// ---- DUTs/EPS Robot/CmdRobot1.TcDUT
{attribute 'qualified_only'}
{attribute 'strict'}
TYPE CmdRobot1 :
(
	noCmd := 0 ,
	Cmd_GoHome:=1 ,
	Cmd_TakePart:=2 ,
	Cmd_PutPart:=4
	//1=回原点程序  2=取料程序  3=放料程序
	
)WORD;
END_TYPE

// ---- DUTs/EPS Robot/DUT_SysFromRobot1.TcDUT
TYPE DUT_SysFromRobot1 :
STRUCT
//Robot-PLC
xHomePosReached	    		:BOOL;//回原点完成
xPickPartPosReached 	  :BOOL;//到达取料位
xPutPartPosReached			:BOOL;//到达放料位
xPickPos1Reached				:BOOL;//到达主流线取料位置1
xPickPos2Reached				:BOOL;//到达主流线取料位置2
xPickPos3Reached				:BOOL;//到达buffer位置取料
xPickTransferPosReached	:BOOL;//到达中转位置
xPutPos1Reached         :BOOL;//到达皮带线位置1
xPutPos2Reached         :BOOL;//到达皮带线位置2
xPutPos3Reached         :BOOL;//到达NG流道位置
xPutPos4Reached					:BOOL;//到达缓存取料位置

xStepRunning						:BOOL;//子程序已运行
xStepRunDone        		:BOOL;//流程已运行
xInitOK            			:BOOL;//初始化完成
xOutofseg1   						:BOOL;//干涉区1外
xOutofseg2          	  :BOOL;//干涉区2外
xOutofseg3          	  :BOOL;//干涉区3外
END_STRUCT
END_TYPE

// ---- DUTs/EPS Robot/DUT_SysToRobot1.TcDUT
TYPE DUT_SysToRobot1 :
STRUCT
//PLC-Robot	
xStepRunPermit      	:BOOL;//流程允许运行
xClampPartDone				:BOOL;//夹取孔板完成	
xReleasePartDone   		:BOOL;//释放孔板完成
xPickPos1Premit				:BOOL;//去主线位置1取料允许
xPickPos2Premit				:BOOL;//去主线位置2取料允许
xPickPos3Premit				:BOOL;//去buffer位置取料允许
xPickTransferPosPremit:BOOL;//去中转位置允许
xPutPos1Premit				:BOOL;//去皮带线位置1放料允许
xPutPos2Premit				:BOOL;//去皮带线位置2放料允许
xPutPos3Premit				:BOOL;//去NG流道位置放料允许
xPutPos4Premit				:BOOL;//去buffer位置放料允许
iMoveMode           	:WORD;//1=回原点   2=取料程序  4=放料程序
iRatio              	:WORD;//机器人速率
END_STRUCT
END_TYPE

// ---- DUTs/EPS Robot/stPutPartPosChoose.TcDUT
{attribute 'qualified_only'}
{attribute 'strict'}
TYPE stPutPartPosChoose :
(
	enum_member := 0,
	CardPositon_1 := 1,
	CardPostion_2 := 2,
	NGPositon	  :=3,
	BufferPostion :=4
)WORD;
END_TYPE

// ---- DUTs/EPS Robot/stTakePartPosChoose.TcDUT
{attribute 'qualified_only'}
{attribute 'strict'}
TYPE stTakePartPosChoose :
(
	enum_member := 0,
	CardPositon_1 := 1,
	CardPostion_2 := 2,
	BufferPostion :=3
)WORD;
END_TYPE

// ---- DUTs/IO/EL1889.TcDUT
TYPE EL1889 :
STRUCT
	INPUT          :word;
END_STRUCT
END_TYPE

// ---- DUTs/IO/EL2889.TcDUT
TYPE EL2889 :
STRUCT
	OUTPUT          :WORD;
END_STRUCT
END_TYPE

// ---- DUTs/Others/DUT_Calibration.TcDUT
TYPE DUT_Calibration :
STRUCT
	strCalibHmi:STRING;	//校准信息
	xWindowsTrigger :BOOL;//窗口调用
	xStartButtonHmi:BOOL;//校准开始按钮
	xNextButtonHmi:BOOL;//下一组
	xCompletedButtonHmi:BOOL;//校准完成按钮
	xNeedCalibration  :BOOL;//需要校准标志位
	iXCounter:INT;//泵头
	iYCounter:INT;//控制器
	rRudongPumpVolume:REAL;//蠕动泵设定量
	rMckVolume			:REAL;//称测量的量
	rDensity				:REAL;//溶液密度
	iType						:INT:=1;//溶液类型
	iInjectCounter	:INT:=1;//注液次数
	xError  			  :BOOL;//报警
	xReset					:BOOL;//复位报警
END_STRUCT
END_TYPE

// ---- DUTs/Others/DUT_Sta.TcDUT
TYPE DUT_Sta :
STRUCT
		Staion:ARRAY[1..gc_uiStationNum] OF  DUT_StaHistory;
END_STRUCT
END_TYPE

// ---- DUTs/Others/DUT_StaHistory.TcDUT
TYPE DUT_StaHistory :
STRUCT
		History:ARRAY [1..500] OF STRING[100];
END_STRUCT
END_TYPE

// ---- DUTs/Others/stEasyPumpsParamter.TcDUT
TYPE stEasyPumpsParamter :
STRUCT
 		xRdyCmd:BOOL;
		xStart:BOOL;
		xReset:BOOL;
		xBusy:BOOL;
		xError:BOOL;
		xDone:BOOL; 
		
		// 手动校准步骤
		iMCalibStep,iOldMCalibStep: INT;

 		iPumpContorller:INT;
		iPumpModule:INT;
		rSetVolume:REAL;
		rRunTime :REAL;
		iCycleNum:INT;
		iBackAngle:INT;
		rAverageRealVolume:REAL;
		arrRealVolume:ARRAY[1..3] OF REAL;
		arrTestRealVolume:ARRAY[1..50] OF REAL;
		arrRecordVolume:ARRAY[1..50] OF REAL;
		iInjectCounter:INT;
		iCalibCounter:INT;
		iRecordCounter:INT;
		//操作
		
		xModulePushStart:BOOL;//单通道注液开始
		xCalibTestStart:BOOL;//校准测试开始
		xRecordDataStart:BOOL;//记录数据开始
		xModulePushOK:BOOL;//注液OK
		xCalibTestOK:BOOL;//校准测试OK
		xRecordDataOK:BOOL;//记录数据OK
		tStableDelay: TON;
		xInitCalibration:BOOL;//初始化校准系数
		xGotoPosition:BOOL;//去校准位置
		xNeedInjectAgain:BOOL;//需要重新注液
		
		//上下偏差
		rESVolume: REAL;//上偏差
		rEIVolume: REAL;//下偏差
		
END_STRUCT
END_TYPE

// ---- DUTs/Others/stWorkStatus.TcDUT
{attribute 'qualified_only'}
{attribute 'strict'}
TYPE stWorkStatus :
(
	None := 0,
	Started:=1,
	Completed:=2
)BYTE;
END_TYPE

// ---- DUTs/Others/tDateAndTime.TcDUT
TYPE tDateAndTime :
STRUCT

     wYear				: WORD;
     wMonth				: WORD;
     wDayOfWeek	    	: WORD;
     wDay				: WORD;
     wHour				: WORD;
     wMinute			: WORD;
     wSecond			: WORD;
     wMilliseconds 	: WORD;

END_STRUCT
END_TYPE

// ---- DUTs/PartData/DUT_BeltLineFixture.TcDUT
TYPE DUT_BeltLineFixture :
STRUCT
 	xMaterialOnOff : BOOL ;
  stProduct : DUT_PartStatus_1 ;
END_STRUCT
END_TYPE

// ---- DUTs/PartData/DUT_LidChecking.TcDUT
TYPE DUT_LidChecking :
STRUCT
	arCameraResult:ARRAY[1..4,1..12] OF INT;
END_STRUCT
END_TYPE

// ---- DUTs/PartData/DUT_MainlineFixture.TcDUT
TYPE DUT_MainlineFixture :
STRUCT
		xMaterialOnOff : BOOL ;
    stProduct : DUT_PartStatus ;
		stProductFlag :DUT_PartFlag;
		stProcessData:DUT_LidChecking;
		arCycletimeStation: ARRAY[1..20] OF REAL;
END_STRUCT
END_TYPE

// ---- DUTs/PartData/DUT_PartFlag.TcDUT
TYPE DUT_PartFlag :
STRUCT
	xLoading_Bypass :BOOL ;
	xLabeling_Bypass: BOOL ;
	xLidExtracting_Bypass : BOOL ;
	xCoverTightening_Bypass : BOOL ;
	xMarking_Bypass: BOOL ;
	xLabelCheck_Bypass: BOOL ;
	xCoverChcek_Bypass:BOOL;
	
	xNeedChangePallet:BOOL;
	xNeedLabelRepeat :BOOL;
END_STRUCT
END_TYPE

// ---- DUTs/PartData/DUT_PartStatus.TcDUT
TYPE DUT_PartStatus :
STRUCT
	xALL_OK : 	BOOL ; //总的OK
	xPart_Normal :BOOL;//产品正常
	xPart_NG	:BOOL;	//其中有NG
	xLoading_OK :BOOL ;
	xLoading_NOK :BOOL;
	xlidInjecting_OK: BOOL ;
	xlidInjecting_NOK :BOOL;
	xLidChecking_OK : BOOL ;
	xLidChecking_NOK :BOOL;
	xAluCovering_OK : BOOL ;
	xAluCovering_NOK :BOOL;
	xAdjusting_OK: BOOL ;
	xAdjusting_NOK :BOOL;
	xCutting_OK		:BOOL;
	xCutting_NOK		:BOOL;
	xEmptying:BOOL;
END_STRUCT
END_TYPE

// ---- DUTs/PartData/DUT_PartStatus_1.TcDUT
TYPE DUT_PartStatus_1 :
STRUCT
	xALL_OK : 	BOOL ; //总的OK
	xPart_Normal :BOOL;//产品正常
	xPart_NG	:BOOL;	//其中有NG
	xCardLoading_OK :BOOL ;
	xCardLoading_NOK :BOOL;
	xBoxLoading_OK: BOOL ;
END_STRUCT
END_TYPE

// ---- DUTs/PartData/DUT_Robot2.TcDUT
TYPE DUT_Robot2 :
STRUCT
		xMaterialOnOff : BOOL ;
        stProduct :ARRAY[1..5] OF DUT_PartStatus ;
END_STRUCT
END_TYPE

// ---- DUTs/PartData/DUT_Process.TcDUT
TYPE DUT_Process :
STRUCT
	xProcessNone				:BOOL;	(*module Process need bypass*)
	xProcessNotStarted     		:BOOL;	(*Module process not start*)
	xProcessStarted          	:BOOL;	(*Module process start*)
	xProcessCompleted     		:BOOL;	(*Module process completed*)
	xQDataCompleted				:BOOL; (*Module data send completed*)
END_STRUCT
END_TYPE

// ---- DUTs/PartSequence/tsPartSequence.TcDUT
TYPE tsPartSequence :
STRUCT
	asSequenceData:ARRAY[0..gc_uiStationNum] OF tsSequence;(*module sequence *)
END_STRUCT
END_TYPE

// ---- DUTs/PartSequence/tsSequence.TcDUT
TYPE tsSequence :
STRUCT
	iSequenceID:INT;(*sequence ID*)
	xRunning:BOOL;(*sequence running*)
	xFinished:BOOL;(*sequence finished*)
	iRequestID:INT;(*request sequence ID initialization value=-1 the program not active *)
	xRequestSucceed:BOOL;(*request sequence succeed*)
	xComplete:BOOL;(*xFinished: true->ack>false*)
	iJobNum:INT; (*program job num*)
	iNumOfParID:INT;(*number of parallel*)
	aiParIDCreated:ARRAY[0..gc_uiStationNum] OF INT;  (*Parallel sequence ID*)
END_STRUCT
END_TYPE

// ---- DUTs/PC/DUT_FomularData.TcDUT
TYPE DUT_FomularData :
STRUCT
	iRotatePosSet:INT;//电动夹爪旋转位置设定
	iRotateSpeSet:INT;//电动夹爪旋转位置旋转速度设定
	iRotateTorSet:INT;//电动夹爪旋转扭力设定
    iClampWPSet:INT;//电动夹爪工作位设定
    iClampMarginSet:INT;//电动夹爪气缸裕量设定
	iCurrentProductModel:INT := 1 ;//当前产品型号
	
	iLiquidInVolumeSet:INT;//加液量
	iLiquidOutVolumeSet:INT;//抽液量
	iLabelStepMotPosSet:INT;//标签机旋转轴旋转角度设定
	iCameraStepMotPosSet:INT;//相机旋转轴旋转角度设定
	
	Rev2:ARRAY[1..10]OF INT;
	

END_STRUCT
END_TYPE

// ---- DUTs/PC/DUT_PCReceive.TcDUT
TYPE DUT_PCReceive :
STRUCT
  iPLCALive : INT ;//保持1s跳动为正常，否则为异常
  iMachineEmptyDone:INT; //1=清空完成  0=无操作
  iLableCompeted:INT;//1=贴标完成
	iInitCommand:INT;//设备初始化命令
	iInitFinished:INT;//设备初始化完成
	iMachineStart:INT;//设备启动
	iShiftOKTotal	:INT;		//	订单OK件计数		
	iShiftNGTotal	:INT;		//	订单NG件计数		
	iRobotUnloadSignal:INT	;//机械手下料信号	1=机械手下料完成   用于计算设备CT
END_STRUCT
END_TYPE

// ---- DUTs/PC/DUT_PCSend.TcDUT
TYPE DUT_PCSend :
STRUCT
	 iPCALive	:INT	;//	心跳	保持1s跳动为正常，否则5s为异常
	 iLableReady	:INT	;//	打印机贴标准备就绪	1=准备就绪  0=未就绪
	 iMachineLampButton	:INT	;//	设备灯控制	1=开灯，0=关灯
	 iInitComfirm	:INT	;//		1=初始化确认  
	 iShiftButton	:INT	;//	订单下发按钮	1=订单下发
	 iMachineEmptyButton	:INT	;//	设备清空按钮	1=设备清空
	 iPCAlarm	:INT	;//	PC报警	1=有报警   0 =无报警
	 iBodyType	:INT	;//	设备产品类型	1…n:分别代表的产品类型
	 iScrapLabel	:INT	;//	废弃空白标签	0=不废弃    1= 废弃空白标签
	 iShiftTotal	:INT	;//	订单总数	订单总数下发
	 iEmptyButtonComfirm:INT;//设备清空确认
END_STRUCT
END_TYPE

// ---- DUTs/PC/DUT_UploadProcessData.TcDUT
TYPE DUT_UploadProcessData :
STRUCT
	iGoodNum:INT ;//良品数
	iNGNum:INT ;//NG数
	iCT:INT ;//总CT
	
    iSTAlarm :ARRAY[1..9] OF DINT; //工站报警字
    iMachineAlarm:DINT ;//设备报警字


    iSTAutoTip: ARRAY[1..9] OF DINT; //工站提示字
    iMachineAutoTip:DINT ;//设备提示字
	
	
	iSTStatus:ARRAY[1..9] OF INT ;//工站状态字
	
	iCoverTightenCT:INT ;//电动夹爪CT
	iCoverTightenRotateCurrentPosition:INT ;//电动夹爪夹持当前位置
	iCoverTightenRotateCurrentSpeed:INT ;//电动夹爪夹持当前速度 
	iCoverTightenRotateCurrentTorque:INT ;//电动夹爪夹持当前扭力

	iPipetCT:INT ;//移液CT
	iLabelCT:INT ;//贴标CT
	iLabelSpeed:INT ;//贴标速度
	Share1:INT;//
	Share2:INT;//
	Share3:INT;//
	Share4:INT;//
	Share5:INT;//
	Share6:INT;//
	Share7:INT;//
	Share8:INT;//
	Share9:INT;//
	Share10:INT;//

END_STRUCT
END_TYPE

// ---- DUTs/Recipe/DUT.TcDUT
TYPE DUT :
STRUCT		
	Length  :INT;
	Width   :REAL;
	Choose  :BOOL;

END_STRUCT
END_TYPE

// ---- DUTs/Recipe/ST_Thermostat.TcDUT
TYPE ST_Thermostat :
STRUCT
	tTON_Delay	:TIME;//热熔时间
END_STRUCT
END_TYPE

// ---- POUs/003_FB/0014_HITBOT/HITBOT_ERROR.TcDUT
{attribute 'qualified_only'}
{attribute 'strict'}
TYPE HITBOT_ERROR :
(
 	NO_ERROR :=0,//无错误
	FLT_PARA :=1,//参数错误
	FLT_READ_PARA:=2,//读取参数错误
	FLT_SET_PARA:=3,//参数设定错误
	FLT_CMD_TIMEOUT:=4,//命令超时
	FLT_RUN_ERROR:=5,//运行报错
	FLT_CONFIGURE_PARA:=6,//配置错误
	FLT_NEED_INIT:=7,//需要先初始化
	FLT_CLAMP_EMPTY:=8//夹空
)INT;
END_TYPE

// ---- POUs/003_FB/0014_HITBOT/stCmdType.TcDUT
{attribute 'qualified_only'}
{attribute 'strict'}
TYPE stCmdType :
(
	iNO_CMD := 0,
	iClamp:=1,
	iRelease:=2,
	iRotateClamp:=3,
	iRotateRelease:=4,
	iRotateRelClamp:=5,
	iRotateRelRelease:=6,
	iInit:=7
	
)INT;
END_TYPE

// ---- POUs/003_FB/0014_HITBOT/stHIBOTLocalPara.TcDUT
TYPE stHIBOTLocalPara :
STRUCT
 	stClampPara  :  stRealPara;//夹持
	stRotateClampPara :  stRealPara;//旋转
	stRotateRelAngle:REAL;//相对旋转角度
END_STRUCT
END_TYPE

// ---- POUs/003_FB/0014_HITBOT/stDeviceStatus.TcDUT
TYPE stDeviceStatus :
STRUCT
 xQStart:BOOL;
 xQRdyCmd:BOOL;
 xQBusy:BOOL;
 xQDone:BOOL;
 xQError:BOOL;
END_STRUCT
END_TYPE

// ---- POUs/003_FB/0014_HITBOT/stOper_Para.TcDUT
TYPE stOper_Para :
STRUCT
 	xHMInitButton , xInitControl : BOOL;
	aHMIClampButton , aHMIReleaseButton , aClampControl , aReleaseControl : ARRAY[1..5] OF BOOL;//夹紧和松开
	aHMIRotateClampButton , aHMIRotateReleaseButton , aRotateClampControl , aRotateReleaseControl : ARRAY[1..5] OF BOOL;//绝对旋转拧紧和松开
	aHMIRotateClampRelButton , aHMIRotateReleaseRelButton , aRotateClampRelControl , aRotateReleaseRelControl : ARRAY[1..5] OF BOOL;//相对旋转拧紧和松开
END_STRUCT
END_TYPE

// ---- POUs/003_FB/0014_HITBOT/stReadPara.TcDUT
TYPE stReadPara :
STRUCT
 rClampPosition:REAL;//夹持位置
 rClampSpeed:REAL;//夹持速度
 rClampCurrent:REAL;//夹持电流

 rRotateAngle:REAL;//旋转角度
 rRotateSpeed:REAL;//旋转速度
 rRotateCurrent:REAL;//旋转电流
 
 rRotateRelAngle:REAL;//相对旋转角度
 
 
 iInitStatus:INT;//0-未初始化  5-初始化完成 其他-初始化中
 iClampStatus:INT;//0 -到位  1-运动中 2-夹持 3-掉落
 iRotateStatus:INT;//0-到位，1-运动中 2-堵转
 rFeedBack_ClampPos	:REAL;//夹持位置反馈
 rFeedBack_ClampSpeed	:REAL;//夹持速度反馈
 rFeedBack_ClampCurrent	:REAL;//夹持电流反馈
 
 rFeedBack_RotatePos	:REAL;//旋转角度反馈
 rFeedBack_RotateSpeed	:REAL;//旋转速度反馈
 rFeedBack_RotateCurrent	:REAL;//旋转电流反馈
 

END_STRUCT
END_TYPE

// ---- POUs/003_FB/0014_HITBOT/stRealPara.TcDUT
TYPE stRealPara :
STRUCT
 	rCurrentSet   		: REAL;//目标力值设置  ( 0.2 - 0.5A )
	rSpeedSet    			: REAL;//运行速度设置  (1-200mm)	
	rPositionSet 		  : REAL;//位置设置值	 (夹持 0-20mm，旋转-36000000-3600000) 
END_STRUCT
END_TYPE

// ---- POUs/003_FB/0014_HITBOT/stSetPara.TcDUT
TYPE stSetPara :
STRUCT
 	aHMIClampPara , aHMIReleasePara : ARRAY[1..5] OF stRealPara;//夹紧轴点位信息
	aHMIRotateClampPara , aHMIRotateReleasePara : ARRAY[1..5] OF stRealPara;//旋转轴点位信息
	aHMIRotateRelClampPara , aHMIRotateRelReleasePara : ARRAY[1..5] OF stRealPara;//旋转轴点位信息
END_STRUCT
END_TYPE

// ---- POUs/003_FB/03_TURINRobotFB/DUTs/CmdRobot.TcDUT
{attribute 'qualified_only'}
{attribute 'strict'}
TYPE CmdRobot :
(
	noCmd                :=0,
	Cmd_GoHome           :=1,//1=回原点 
	Cmd_GoAutoProcesses  :=2//到取料位
)INT;
END_TYPE

// ---- POUs/003_FB/03_TURINRobotFB/DUTs/DUT_SysFromRobot.TcDUT
TYPE DUT_SysFromRobot :
STRUCT
//Robot-PLC
xEstop,   			      //机器人急停
xLocal_Remote,			  //本地/远程
xEnable,              //机器人使能
xRuntip,              //运行中
xStopTip,             //停止
xAt_HomePosition,     //在原点位
xAt_PickPoint,        //在取料位
xAt_PickPointUp,      //在取料位上方
xAt_PutPoint1,        //在放料位1
xAt_PutPoint2,        //在放料位2
xAt_PutPoint3,        //在放料位3
xStepRuning,          //流程运行中
xInitOK,              //初始化完成
xGoHomeDone,          //回原点完成
xOutofseg1,           //取料区域
xOutofseg2,           //放料区域
xSeg1Complete,           
xSeg2Complete,
xOutofseg3,           
xCycleDone      :BOOL;//循环完成
END_STRUCT
END_TYPE

// ---- POUs/003_FB/03_TURINRobotFB/DUTs/DUT_SysToRobot.TcDUT
TYPE DUT_SysToRobot :
STRUCT
//PLC-Robot	
xStepRunPermit,            //流程允许运行
xGo_PickPoint,             //到取料位
xGo_PickPointUp,           //到取料位上方
xGo_PutPoint1,             //到放料位1
xGo_PutPoint2,             //到放料位2
xGo_PutPoint3,             //到放料位3
xGo_StandByPos,            //回待机点
xResetWorkDone,            //复位工作完成
xGo_PutPoint11,             //到放料位11
xGo_PutPoint12,             //到放料位12
xGo_PutPoint13       :BOOL; //到放料位13

iMoveMode           :WORD;//1=回原点 2=自动流程 
iRatio              :WORD;//机器人速率

END_STRUCT
END_TYPE

// ---- POUs/003_FB/03_TURINRobotFB/DUTs/ST_Sys_Para.TcDUT
TYPE ST_Sys_Para :
STRUCT
	strSlaveIP				: STRING(15) := '127.0.0.0';	//modbus子站IP地址
	iSlavePort				: UINT := 502;					//默认是502
	bySlaveID 				: BYTE;							//modbus rtu子站地址
END_STRUCT
END_TYPE

// ---- POUs/003_FB/03_TURINRobotFB/DUTs/ST_TURINROBOT_Data.TcDUT
TYPE ST_TURINROBOT_Data :
STRUCT		
	i_Ready:               BOOL;				
	i_Running:             BOOL;				
	i_Paused:              BOOL;				
	i_Error:               BOOL;				
	i_EStopOn:             BOOL;							
	i_SError:              BOOL;				
	i_Waning:              BOOL;			
	i_MotorsOn:            BOOL;												
	i_AutoMode:            BOOL;				
  i_TeachMode:           BOOL;
	i_CmdError:            BOOL;					
				
  o_Start:               BOOL;	
  o_Init:                BOOL;							
	o_Stop:                BOOL;			
	o_Pause:               BOOL;				
	o_Continue:            BOOL;				
	o_Reset:               BOOL;				
	o_SetMotorsOn:         BOOL;			
	o_SetMotorsOff:        BOOL;	
	o_RunCondition:        BOOL;				

END_STRUCT
END_TYPE

// ---- POUs/003_FB/03_TURINRobotFB/DUTs/TURIN_ERROR.TcDUT
{attribute 'qualified_only'}
{attribute 'strict'}
TYPE TURIN_ERROR :
(
	NO_ERROR 								:= 0,	
  FLT_SYSREADY             := 1000, (*系统没有准备好*)
  FLT_AUTOMODE             := 1001, (* 机器人没有处于自动状态*)
  FLT_PROMERROR            := 1002, (* 启动主程序错误*)
	FLT_PARA                 := 1003, (* 启动主程序错误*)
	
  FLT_CMDERROR             := 1010, (*指令你执行错误*)
  FLT_SERROR               := 1011, (* 系统错误发生 *)
  FLT_ESTOPON              := 1012, (*急停触发*)
	FLT_ERROR                := 1013, (*有错误发生*)  
	FLT_CONNECTERROR         := 1014, (*有错误发生*)  
  FLT_NO_INIT              := 1015,(* 没有初始化完成 *)   
	FLT_INIT_TIMEOUT         := 1016,(* 没有初始化完成 *)   
	FLT_Warning       			 := 1017,(* 机械手警告 *)  
	FLT_No_Runing             :=1018(*机器人没有运行*)
)INT;
END_TYPE

// ---- POUs/003_FB/03_TURINRobotFB/DUTs/TURIN_STATE.TcDUT
{attribute 'qualified_only'}
{attribute 'strict'}
TYPE TURIN_STATE :
(
	DORMANT  							:= 0,
	EXECUTING 						:= 1,
	DONE 								  := 2,
	INERROR								:= 3,
	ABORTING 							:= 4,
	ABORTED 							:= 5,
	RESETING 							:= 6
);
END_TYPE

// ---- POUs/003_FB/03_TURINRobotFB/DUTs/T_MaxString.TcDUT
TYPE T_MaxString : string(255); END_TYPE

// ---- POUs/003_FB/05_StationFB/E_State.TcDUT

{attribute 'strict'}
TYPE E_State :
(
	NotReady:=0,				//未准备好
	iRunning:=3,					//运行中
	Alarm:=2,					//报警中
	Ready:=1,					//准备好
	Done:=4          //工站完成
	
)UINT;
END_TYPE

// ---- POUs/003_FB/0009_MKC204C/DUTs/MT_MCK_CMD.TcDUT
{attribute 'qualified_only'}
{attribute 'strict'}
TYPE MT_MCK_CMD :
(
 	Nodef,
	Cmd_SerialNum,//获取序列号,I4
	Cmd_Shelling,//稳态去皮重,T
	Cmd_ShellingInstanly,//立即去皮重,TI	
	Cmd_SetTare,//预置皮重，TA
	Cmd_ClearTare,//清除皮重,TAC
	Cmd_ClearZero,//稳态清零,Z
	Cmd_ClearZeroInstanly,//立即清零,ZI
	Cmd_AcquireWeight_Steady,//单次获取稳态重量,S
	Cmd_AcquireWeight_RealTime,//连续获取重量,SI
	Cmd_AcquireWeight_Continuous,//连续获取重量,SIR
	Cmd_AcquireWeight_Stop,//中断连续获取重量,SI
	Cmd_Restart	//重启秤体
);
END_TYPE

// ---- POUs/003_FB/0009_MKC204C/DUTs/MT_MCK_ERROR.TcDUT
{attribute 'qualified_only'}
{attribute 'strict'}
TYPE MT_MCK_ERROR :
(
 	No_ERROR := 0,	
  	FLT_PARA             			  	:= 1, (* E-Gripper Parameter fault   程序配置参数有问题 *)
  	FLT_CONNECT       		        	:= 2, (* E-Gripper not ready 旋转有通信报警*)  
  	FLT_RDYCMD           			    := 3, (* E-Gripper read/write command while not ready 预留*)  
  	FLT_STOP_TIMEOUT 					:= 12, (* E-Gripper org command execute Timeout *)  
	FLT_CMD_TIMEOUT    		 			:= 15, (* E-Gripper release command execute Timeout *) 
  	FLT_LogicaL     					:= 17, (* 逻辑错误 *)  
 	FLT_Syntax     						:= 18, (* 语言错误 *) 
 	FLT_CommandCantSend     			:= 19, (* 命令不能发送 *) 
  	FLT_Par     						:= 20, (* 参数错误 *) 
  	FLT_ZI     							:= 21, (* 清零未响应 *) 
  	FLT_ZOverMax     					:= 22, (* 清零超出上限 *) 	
  	FLT_ZOverMin     					:= 23,(* 清零低于上限 *)
  	FLT_CmdFeedback     				:= 24,(* 指令反馈错误 *)	
  	FLT_TOverMax     					:= 25, (* 去皮超出上限 *) 	
  	FLT_TOverMin     					:= 26,(* 去皮低于上限 *)	
		FLT_CannotExecutable			:=27,(*理解指令，但不能执行*)
		FLT_SIROverMIN						:=28,(*重复读取超出下限*)
		FLT_SIROverMAX						:=29,(*重复读取超出上限*)
		FLT_SIRERROR						 :=30(*重复读取报错*)
)INT;
END_TYPE

// ---- POUs/003_FB/0009_MKC204C/DUTs/ST_DeviceOpe.TcDUT
{attribute 'qualified_only'}
{attribute 'strict'}
TYPE ST_DeviceOpe :
STRUCT
	xReadSerialNum_HMI,xReadSerialNum_Auto							:BOOL;//获取序列号,I4
	xShelling_HMI,xShelling_Auto									:BOOL;//稳态去皮重,T
	xShellingInstanly_HMI,xShellingInstanly_Auto					:BOOL;//立即去皮重,TI	
	xSetTare_HMI,xSetTare_Auto										:BOOL;//预置皮重，TA
	xlearTare_HMI,xlearTare_Auto									:BOOL;//清除皮重,TAC
	xClearZero_HMI,xClearZero_Auto									:BOOL;//稳态清零,Z
	xClearZeroInstanly_HMI,xClearZeroInstanly_Auto					:BOOL;//立即清零,ZI
	xAcquireWeight_Steady_HMI,xAcquireWeight_Steady_Auto			:BOOL;//单次获取稳态重量,S
	xAcquireWeight_RealTime_HMI,xAcquireWeight_RealTime_Auto		:BOOL;//连续获取重量,SI
	xAcquireWeight_Continuous_HMI,xAcquireWeight_Continuous_Auto	:BOOL;//连续获取重量,SIR
	xAcquireWeight_Stop_HMI,xAcquireWeight_Stop_Auto				:BOOL;//中断连续获取重量,SI
	xRestart_HMI,xRestart_Auto										:BOOL;//重启秤体	
	xRepeatRead_Hmi,xRepeatRead_Auto							:BOOL;//重复读取重量
END_STRUCT
END_TYPE

// ---- POUs/003_FB/0009_MKC204C/DUTs/ST_MCK_ParOut.TcDUT
{attribute 'qualified_only'}
{attribute 'strict'}
TYPE ST_MCK_ParOut :
STRUCT
	sSrialNumber		:STRING;//序列号
	rCurrentWeight		:REAL;//当前重量
	rCurrentTareWight	:REAL;//当前皮重
	rWeightMax			:REAL;//最大称重值
	rWeightMin			:REAL;//最小称重值	
	sWeightUnit			:STRING;//单位
	sErrorID			:STRING;//报错内容
	xContinuesRead	:BOOL;//连续读取重量中
	rStableWeight	:REAL;//稳态重量记录
	rRepeatWeight:REAL;//循环读取中
END_STRUCT
END_TYPE

// ---- POUs/003_FB/0009_MKC204C/DUTs/ST_SysPar.TcDUT
{attribute 'qualified_only'}
{attribute 'strict'}
TYPE ST_SysPar :
STRUCT
	sRemoteHost			: T_IPv4Addr ;
	nRemotePort			: UINT := 0;    
	bySlaveID 			: BYTE;	
END_STRUCT
END_TYPE

// ---- POUs/003_FB/0010_LoadCell/DUT_DeviceOpe.TcDUT
TYPE DUT_DeviceOpe :
STRUCT
	xReadGROSSHmi,xReadGROSSAuto							:BOOL;//读取总值GROSS
	//xReadNETHmi,xReadNETAuto									:BOOL;//读取净值NET
	//xReadPEAKHmi,xReadPEAKAuto								:BOOL;//读取峰值PEAK
	//xReadPVHmi,xReadPVAuto										:BOOL;//读取峰-谷值P-V
	//xReadDISPHmi,xReadDISPAuto								:BOOL;//读取显示值
	xSetZEROHmi,XSetZEROAuto									:BOOL;//设定零点
	xSetZEROSaveHmi,xSetZEROSaveAuto					:BOOL;//保存零点
END_STRUCT
END_TYPE

// ---- POUs/003_FB/0012_EasyPump/DUT/PumpError.TcDUT
{attribute 'qualified_only'}
{attribute 'strict'}
TYPE PumpError :
(
 	NO_ERROR :=0,//无错误
	FLT_PARA :=1,//参数错误
	FLT_FLUVOLUM_TIME_PARA:=2,//时间参数错误
	FLT_READ_PARA:=3,//读取参数错误
	FLT_SET_PARA:=4,//参数设定错误
	FLT_CMD_TIMEOUT:=5,//命令超时
	FLT_RUN_ERROR:=6,//运行报错
	FLT_Calib_OverFlow:=7,//误差过大
	FLT_CALIB_PARA:=8,//校准参数设定错误
	FLT_CONFIGURE_PARA:=9//配置错误
);
END_TYPE

// ---- POUs/003_FB/0012_EasyPump/DUT/stEasyPumpHeadType.TcDUT
{attribute 'qualified_only'}
{attribute 'strict'}
TYPE stEasyPumpHeadType :
(
	i_MiniPump01:=1,
	i_MiniPump02:=2,	
	
	i_HandyPump01:=3,
	i_HandyPump02:=4,	
	
	i_EasyPumpI_III:=5,//单通道
	i_EasyPumpII_IV:=6,//单通道
	i_EasyPumpV_VI:=7,//双通道

	i_AMC1_AMC12:=8,//适用(内径x壁厚0.13-3/0.8-1mm)
	i_YZ1515x:=9,//适用13#,14#,16#,17#,18#,19#,25#管
	i_YZ2515x:=10,//适用15#,24#管	
	
	iDY15:=11,//
	iDY25:=12,
	
	iUD15:=13
)INT;
END_TYPE

// ---- POUs/003_FB/0012_EasyPump/DUT/stEasyPumpHmi.TcDUT
TYPE stEasyPumpHmi :
STRUCT
	xPush_Hmi,xPush_Auto 										: ARRAY[1..5] OF BOOL;
	xPull_Hmi,xPull_Auto 										: ARRAY[1..5] OF BOOL;	
	xStop_Hmi,xStop_Auto 										: BOOL;
	xFullSpeedPush_Hmi,xFullSpeedPush_Auto 	: BOOL;
	xFullSpeedPull_Hmi,xFullSpeedPull_Auto 	: BOOL;
	xFullSpeedStop_Hmi,xFullSpeedStop_Auto 	: BOOL;
	xModulePush_Hmi,xModulePush_Auto		 		: BOOL;	
	xCalibAction_Hmi,xCalibAction_Auto : BOOL;
	xCalibInit_Hmi,xCalibInit_Auto					: BOOL;	
	xAdjust_Hmi,xAdjust_Auto			: BOOL;
END_STRUCT
END_TYPE

// ---- POUs/003_FB/0012_EasyPump/DUT/stEasyPumpSoftType.TcDUT
{attribute 'qualified_only'}
{attribute 'strict'}
TYPE stEasyPumpSoftType :
(
	i_P13:=1,//13#软管,0.8x1.6
	i_P14:=2,//14#软管,1.6x1.6
	i_P15:=15,//15#软管,1.6x1.6
	i_P19:=3,//19#软管,2.4x1.6
	i_P16:=4,//16软管,3.1x1.6
	i_P25:=5,//25#软管,4.8x1.6	
	i_P1_1:=6,//1x1#软管,1x1
	i_P2_1:=7,//2x1#软管,2x1
	i_P2_5_1:=8,//2.5x1#软管,2.5x1	
	i_P3_1:=9,//3x1#软管,3x1
	i_P17:=10,//17#软管,6.4x1.6		
	i_P18:=11,//18#软管,7.9x1.6	
	i_P24:=12,//24#软管,6.4x2.4		
	i_P35:=13,//34#软管,7.9x2.4
	i_P36:=14//36#软管,9.6x2.4
)INT;
END_TYPE

// ---- POUs/003_FB/0012_EasyPump/DUT/stEasyPumpType.TcDUT
{attribute 'qualified_only'}
{attribute 'strict'}
TYPE stEasyPumpType :
(
	i_LabV:=1,//LabV系列
	i_LabF1:=2,//0.1-150rpm
	i_LabF3:=3,//0.1-350rpm	
	i_LabF4:=4,//0.1-600rpm	
	i_F:=5,//F系列
	i_M:=6,//M系列
	i_V:=7,//V系列
	i_BT_D:=8,//BT_D系列	
	i_PDS:=9,//PDS系列	,五位蠕动泵	
	i_DFPluse:=10//DFPluse系列
)INT;
END_TYPE

// ---- POUs/003_FB/0012_EasyPump/DUT/stOperType.TcDUT
{attribute 'qualified_only'}
{attribute 'strict'}
TYPE stOperType :
(
 	iWait:=0,
	iPush := 1,
	iPull :=2,
	iModulePush:=3,
	iStop:=4,
	iFullSpeedPush:=5,
	iFullSpeedPull:=6,
	iFullSpeedStop:=7,
	iCalibAction:=8,
	iCalibInit:=9,
	iAdjust:=10
)INT;
END_TYPE

// ---- POUs/003_FB/0012_EasyPump/DUT/st_EasyPump.TcDUT
TYPE st_EasyPump :
STRUCT
 iPumpType:INT;//泵头类型
 iHosePipeType:INT;//软管类型
END_STRUCT
END_TYPE

// ---- POUs/003_FB/0012_EasyPump/DUT/ST_StepStatus.TcDUT
TYPE ST_StepStatus :
STRUCT
 xStart:BOOL;
 xBusy:BOOL;
 xDone:BOOL;
 xError:BOOL;
END_STRUCT
END_TYPE

// ---- POUs/003_FB/0012_EasyPump/DUT/ST_LocalPara.TcDUT
TYPE ST_LocalPara :
STRUCT
	rFluVolumeSet   : REAL;//液量设定 0.0-99999.0 mL(0.1ml)
	rRuntimeSet     : REAL;//运行时间设定 0.1-9999s(0.1s)
	iCycleNumber		: INT;//重复次数
	iModuleAdress		: INT;//灌装单元地址
	iModuleSpeed		: REAL;//灌装单元速度
	iModuleRealVolume	: REAL;//灌装实际液量	
	iDirectionSet:INT;//方向
	rVirualTime			:REAL;//虚假的时间
  iAccuracySet				:REAL;//精度要求，如果是4%请填写0.04
	iBackAngle:INT;//回吸角度  0-360
END_STRUCT
END_TYPE

// ---- POUs/003_FB/0012_EasyPump/DUT/ST_ReadPara.TcDUT
TYPE ST_ReadPara :
STRUCT
 rFluVolume:REAL;//显示液量
 rRuntime:REAL;//显示运行时间
 iDirectionSet:INT;//显示方向
 iCycleNumber		: INT;//重复次数
 iModuleAdress:INT;//显示单元
 iRunning:INT;//显示是否在运行
 iBackAngle:INT;//显示回吸角度
END_STRUCT
END_TYPE

// ---- POUs/003_FB/0012_EasyPump/DUT/ST_SetPara.TcDUT
TYPE ST_SetPara :
STRUCT
 	rPullFluVolume			:ARRAY[1..5] OF  REAL;//液量设定 0.0-99999.0 mL(0.1ml)
	rPushFluVolume			:ARRAY[1..5] OF  REAL;//液量设定 0.0-99999.0 mL(0.1ml)	
	rPullRuntime			:ARRAY[1..5] OF  REAL;//运行时间设定 0.1-9999s(0.1s)
	rPushRuntime			:ARRAY[1..5] OF  REAL;//运行时间设定 0.1-9999s(0.1s)	
	iPullBackAngle		:ARRAY[1..5] OF  INT;//回吸角度
	iPullCycleNumber		:ARRAY[1..5] OF  INT;//重复次数	
	iPushCycleNumber		:ARRAY[1..5] OF  INT;//重复次数	
	iPushBackAngle			:ARRAY[1..5] OF INT;//回吸角度
	iDirectionSet				:INT;//方向设定
	iAccuracySet				:REAL;//精度要求，如果是4%请填写0.04
	
	iPumpType					: RudongPump_PumpType;//泵类型选择
	iPumpTypeSet				: RudongPump_PumpHeadType;//泵头类型
	iHosePipeTypeSet			: RudongPump_SoftPipeType;//软管类型	
	
	iModuleAdress		:INT;//灌装单元地址
	rModuleSpeed		:REAL;//灌装单元速度
	rModuleRealFluVolume:REAL;//实际灌装量
	rCalFluVolume		:REAL;//校准液量
	rCalTime			:REAL;//校准时间
	rCalNum				:INT;//校准加液次数	
	rCalBackAngle:INT;//校准回吸角度
	
	rSpeedRatio  : REAL:=2.733;//根据泵头软管型号不同有变化
END_STRUCT
END_TYPE

// ---- POUs/003_FB/10_CylinderFB/ST_DataCylinder.TcDUT
TYPE ST_DataCylinder :
STRUCT
	tHP_Delay					 : TIME ;					//原点延时
	tWP_Delay					 : TIME ;					//动点延时
	Alarm_Delay					: TIME := t#5s;					//报警延时
END_STRUCT
END_TYPE

// ---- POUs/003_FB/0013_RGI_14_new/RGI_14_ERROR.TcDUT
TYPE RGI_14_ERROR :
(
	NO_ERROR := 0,
	/// E-Gripper 参数配置有错误
	FLT_PARA := 1,
	/// E-Gripper not ready 有通信报警
	FLT_CONNECT := 2,
	/// E-Gripper read/write command while not ready 预留
	FLT_RDYCMD := 3,
	///驱动器报警
	FLT_DEVICE_ERROR := 4,
	///没有上电
	FLT_POWERON := 5,
	/// E-Gripper 夹紧超时 
	FLT_CLAMP_TIMEOUT := 10,
	/// E-Gripper 松开超时 
	FLT_ROTATE_TIMEOUT := 11,
	/// E-Gripper 回原点超时 
	FLT_ORG_TIMEOUT := 12,
	/// E-Gripper 夹紧指令执行超时 
	FLT_CLAMPCMD_TIMEOUT := 13,
	/// E-Gripper 松开指令执行超时 
	FLT_ROTATECMDABS_TIMEOUT := 14,
	/// E-Gripper 松开指令执行超时 
	FLT_ROTATECMDREF_TIMEOUT := 17,
	/// E-Gripper 回原点指令执行超时 
	FLT_ORGCMD_TIMEOUT := 15,
	///物体掉落
	FLT_CLAMP_DROP := 16,
	/// E-Gripper reference not OK 没有回原点过程中执行指令
	FLT_xRefOk := 20,
	/// E-Gripper Clamp Para error 发送夹紧参数错误
	FLT_CLAMP_PARA := 21,
	/// E-Gripper 松开指令超时
	FLT_ClAMP_RELEASEFAIL := 24,
	/// E-Gripper 夹紧物体失败 
	FLT_ClAMP_CLAMPFAIL := 25,
	/// E-Gripper 关盖失败
	FLT_ROTATE_CLAMPFAIL := 26,
	/// E-Gripper 开盖失败 
	FLT_ROTATE_RELEASEFAIL := 27
);
END_TYPE

// ---- POUs/003_FB/0013_RGI_14_new/ST_RGI_14_Sys_Para.TcDUT
TYPE ST_RGI_14_Sys_Para :
STRUCT
	///modbus子站IP地址
	strSlaveIP: STRING(15) := '127.0.0.0';
	///默认是502
	iSlavePort: UINT := 502;
	///modbus rtu子站地址		
	bySlaveID: BYTE;
END_STRUCT
END_TYPE

// ---- POUs/003_FB/0013_RGI_14_new/ST_RGI_HMIStates.TcDUT
TYPE ST_RGI_HMIStates :
STRUCT
	///完成条件满足
	xDone: BOOL;
	///动作正在执行
	xBusy: BOOL;
	///指令被打断
	xAborted: BOOL;
	///错误条件满足
	xError: BOOL;
	///错误码
	eErrorID: RGI_14_ERROR;
	///eMobbusErrorID: MODBUS_ERROR;//modubs 报警信息
	xRdyCmd: BOOL;
	xRefOk: BOOL;
	eClampActCmd: RGI_14_CMD;
	///0：运动中，1：到达位置；2：夹住物体；3：物体掉落
	iClampStatus: INT;
	///夹爪夹空
	xGripClampEmpty: BOOL;
	///掉落发生
	xDropOccur: BOOL;
	///关盖失败
	xClosecoverFailure: BOOL;
	///开盖失败
	xOpencoverFailure: BOOL;
	sHmiError: STRING;
END_STRUCT
END_TYPE

// ---- POUs/003_FB/0013_RGI_14_new/ST_RGI_Opera.TcDUT
TYPE ST_RGI_Opera :
STRUCT
	///初始化控制
	xHMInitButton: BOOL;
	///初始化控制
	xInitControl: BOOL;
	///夹爪控制
	aHMIClampButton: ARRAY[1..10] OF BOOL;
	///夹爪控制
	aHMIReleaseButton: ARRAY[1..10] OF BOOL;
	///夹爪控制
	aClampControl: ARRAY[1..10] OF BOOL;
	///夹爪控制
	aReleaseControl: ARRAY[1..10] OF BOOL;
	///绝对旋转控制
	aHMIRotateClampButton: ARRAY[1..10] OF BOOL;
	///绝对旋转控制
	aHMIRotateReleaseButton: ARRAY[1..10] OF BOOL;
	///绝对旋转控制
	aRotateClampControl: ARRAY[1..10] OF BOOL;
	///绝对旋转控制
	aRotateReleaseControl: ARRAY[1..10] OF BOOL;
	///相对旋转控制	
	aHMIRotateClampRefButton: ARRAY[1..10] OF BOOL;
	///相对旋转控制	
	aHMIRotateReleaseRefButton: ARRAY[1..10] OF BOOL;
	///相对旋转控制	
	aRotateClampRefControl: ARRAY[1..10] OF BOOL;
	///相对旋转控制	
	aRotateReleaseRefControl: ARRAY[1..10] OF BOOL;
	xHMIReset: BOOL;
	xHMIPower: BOOL;
	///测试模式时候不做NG检测
	xTestMode: BOOL;
END_STRUCT
END_TYPE

// ---- POUs/003_FB/0013_RGI_14_new/ST_RGI_PosPara.TcDUT
TYPE ST_RGI_PosPara :
STRUCT
	///夹紧轴夹紧力设置
	aHMIClampiTorqueSet: ARRAY[1..10] OF INT;
	///夹紧轴夹紧力设置
	aHMIReleasepiTorqueSet: ARRAY[1..10] OF INT;
	///夹紧轴夹紧速度设置	
	aHMIClampiSpeedSet: ARRAY[1..10] OF INT;
	///夹紧轴夹紧速度设置	
	aHMIReleasepiSpeedSet: ARRAY[1..10] OF INT;
	///夹紧轴夹紧角度设置	
	aHMIClampiPosAngleSet: ARRAY[1..10] OF INT;
	///夹紧轴夹紧角度设置	
	aHMIReleasepiPosAngleSet: ARRAY[1..10] OF INT;
	///旋转轴旋转力设置	
	aHMIRotateiTorqueSet: ARRAY[1..10] OF INT;
	///旋转轴旋转力设置	
	aHMIRotateReleaseiTorqueSet: ARRAY[1..10] OF INT;
	///旋转轴旋转速度设置	
	aHMIRotateClampiSpeedSet: ARRAY[1..10] OF INT;
	///旋转轴旋转速度设置	
	aHMIRotateReleaseiSpeedSet: ARRAY[1..10] OF INT;
	///旋转轴旋转角度设置	
	aHMIRotateClampiPosAngleSet: ARRAY[1..10] OF INT;
	///旋转轴旋转角度设置	
	aHMIRotateReleaseiPosAngleSet: ARRAY[1..10] OF INT;
	///旋转轴相对旋转力设置	
	aHMIRotateRefiTorqueSet: ARRAY[1..10] OF INT;
	///旋转轴相对旋转力设置	
	aHMIRotateReleaseRefiTorqueSet: ARRAY[1..10] OF INT;
	///旋转轴相对旋转速度设置	
	aHMIRotateClampRefiSpeedSet: ARRAY[1..10] OF INT;
	///旋转轴相对旋转速度设置	
	aHMIRotateReleaseRefiSpeedSet: ARRAY[1..10] OF INT;
	///旋转轴相对旋转角度设置	
	aHMIRotateClampRefiPosAngleSet: ARRAY[1..10] OF INT;
	///旋转轴相对旋转角度设置	
	aHMIRotateReleaseRefiPosAngleSet: ARRAY[1..10] OF INT;
END_STRUCT
END_TYPE

// ---- POUs/003_FB/14_MachineFB/ST_DataMachine.TcDUT
TYPE ST_DataMachine :
STRUCT
	bDummyDisabled				: BOOL;					//点检屏蔽
	nSampleSet					: UINT;					//取样数量设置
	rMasterSpeed                : REAL;                 //主轴送料速度mm/s
	rCycleTime					: REAL;					//循环时间，单位s
	nGoods						: UDINT;				//当前良品数量
	nBads						: UDINT;				//当前不良数量
	nTotal						: UDINT;				//当前总数量
	rYield						: REAL;					//当前良品率
	rReject						: REAL;					//当前不良率
	nTotalGoods					: UDINT;				//历史良品数量
	nTotalBads					: UDINT;				//历史不良数量
	nTotalOutputs				: UDINT;				//历史总数量
	rTotalYield					: REAL;					//历史良品率
	rTotalReject				: REAL;					//历史不良率
	nRunningTimer				: UDINT;				//运行时间计时器，单位100ns，除以10000单位ms
	nRunningTime				: UDINT;				//运行时间总秒数
	nRunningDays				: UDINT;				//运行时间-天
	nRunningHour				: UINT;					//运行时间-时
	nRunningMinute				: UINT;					//运行时间-分
	nRunningSecond				: UINT;					//运行时间-秒
END_STRUCT
END_TYPE

// ---- POUs/003_FB/14_MachineFB/ST_OpeButton.TcDUT
TYPE ST_OpeButton :
STRUCT
	xStart						: BOOL;					//启动按钮
	xStop						: BOOL;					//停止按钮
	xReset						: BOOL;					//复位按钮
	xPause						: BOOL;					//暂停按钮
	xInit						: BOOL;					//初始化按钮
	xManualMode					: BOOL;					//手动模式
	xAutoMode					: BOOL;					//自动模式



END_STRUCT
END_TYPE

// ---- POUs/003_FB/19-AxisFB/DUT_ActPos.TcDUT
TYPE DUT_ActPos :
STRUCT
		Mode :UINT:=1;
		Pos:REAL:=1.0;
		
END_STRUCT
END_TYPE

// ---- POUs/003_FB/19-AxisFB/ST_DataAxis.TcDUT
TYPE ST_DataAxis :
STRUCT
	rJogVelocity				: REAL:=1;				//轴Jog速度
	rAcceleration,rDeceleration : REAL ;
	rRelativeDistance,rRelativeVelocity,rVelocityVel      : REAL ;
	rManualVelocity			: REAL:=10;				//轴手动速度
	rAutoVelocity				: REAL:=50;				//轴自动速度
	rMovePosition				: ARRAY[1..gc_uiAxisMoveNum] OF REAL;//绝对定位位置
	rMoveVelocity				: ARRAY[1..gc_uiAxisMoveNum] OF REAL;//绝对定位速度
	tInPosition					: ARRAY[1..gc_uiAxisMoveNum] OF TIME;//绝对到位延时
END_STRUCT
END_TYPE

// ---- POUs/003_FB/41_GetSystemTime/DUT_TIMESET.TcDUT
TYPE DUT_TIMESET :
STRUCT

	sTempTimeYYMMDD: STRING;
	sTempTimeHO: STRING;
	sTempTimeMI: STRING;
	sTempTimeSe: STRING;
END_STRUCT
END_TYPE

// ---- POUs/003_FB/0016_Recipe/ST_Recipe.TcDUT
TYPE ST_Recipe :
STRUCT
	Axis						: ARRAY[1..gc_uiAxisNum] OF ST_DataAxis;
	Cylinder					: ARRAY[1..gc_uiCylinderNum] OF ST_DataCylinder;
	RGI14                  		: ARRAY[1..gc_uiRGI_14_Number] OF ST_RGI_PosPara;
	RudongPump					: ARRAY[1..gc_uiRudongPump]OF RudongPump_RunData;//蠕动泵参数
	Thermostat					:ARRAY[1..gc_uiPXF5Num] OF ST_Thermostat;
	ERG20						:ARRAY[1..gc_uiHITBOT_Number] OF ST_Huiling_Pers_Para;
	TURIN						:ARRAY[1..gc_uiTURINRobot_Num] OF ST_TURINROBOT_Data;
	Camera						:ARRAY[1..gc_uiCameraNum] OF ST_CameraPara;
   TimeS						:ARRAY[1..10] OF TIME;//[1]-贴标延时
	 EasyPumps					:ARRAY[1..gc_uiRudongPump] OF ST_SetPara;
	 ERG20C					:ARRAY[1..gc_uiHITBOT_Number] OF stSetPara;	
END_STRUCT
END_TYPE

// ---- POUs/003_FB/53_RudongPump/08_PeristalticPumpFB/DUTs/RudongPump_CMD.TcDUT
{attribute 'qualified_only'}
{attribute 'strict'}
TYPE RudongPump_CMD ://只有一个夹紧轴
(
  Nodef,
	Cmd_Configure,//配置指令（泵头和软管指令）
  	Cmd_Push,//注液指令
	Cmd_Pull,//吸液指令 
 	 Cmd_Stop,//停止指令
	Cmd_FullSpeedPush,//全速启动
	Cmd_FullSpeedPull,//全速启动
	Cmd_FullSpeedStop,//全速停止
	Cmd_CalPump,//校准泵头
	Cmd_CalReset,//校准泵头
	Cmd_CalParWrite	//校准参数写入
);
END_TYPE

// ---- POUs/003_FB/53_RudongPump/08_PeristalticPumpFB/DUTs/RudongPump_ERROR.TcDUT
{attribute 'qualified_only'}
{attribute 'strict'}
TYPE RudongPump_ERROR :
(
	No_ERROR := 0,
	/// E-Gripper Parameter fault   程序配置参数有问题 
	FLT_PARA := 1,
	/// E-Gripper not ready 旋转有通信报警
	FLT_CONNECT := 2,
	/// E-Gripper read/write command while not ready 预留
	FLT_RDYCMD := 3,
	/// 配置参数错误 
	FLT_CONFIGURE_PARA := 4,
	/// 流量时间配置错误 
	FLT_FLUVOLUM_TIME_PARA := 5,
	/// E-Gripper release  execute Timeout 
	FLT_PUSH_TIMEOUT := 10,
	/// E-Gripper org  execute Timeout 
	FLT_PULL_TIMEOUT := 11,
	/// E-Gripper org command execute Timeout 
	FLT_STOP_TIMEOUT := 12,
	/// E-Gripper org command execute Timeout 
	FLT_FULLSPEEDSTOP_TIMEOUT := 13,
	/// E-Gripper org command execute Timeout 
	FLT_FULLSPEEDSTART_TIMEOUT := 14,
	/// E-Gripper release command execute Timeout 
	FLT_CMD_TIMEOUT := 15,
	/// E-Gripper release command execute Timeout 
	FLT_RUN_FALL := 16,
	/// E-Gripper org  execute Timeout 
	FLT_PumpCal_TIMEOUT := 17,
	/// E-Gripper org  execute Timeout 
	FLT_PumpCal_OverFlow := 18,
	/// Modbus 
	FLT_Mobdus := 19
	
)INT;
END_TYPE

// ---- POUs/003_FB/53_RudongPump/08_PeristalticPumpFB/DUTs/RudongPump_IOData.TcDUT
TYPE RudongPump_IOData :
STRUCT
	//夹紧轴输出
	O_PumpType           : INT;//泵头型号(0-8)
	O_HosePipeType       : INT;//软管型号
	O_ControlSet         : INT;//启停控制；1（启动）;0(停止)
	O_DirectionSet       : INT;//方向控制：1（顺时针）;0（逆时针）
	O_FullSpeedControl   : INT;//全速运行: 1：启动全速; 0：停止全速
	O_FluVolumeSet       : REAL;//液量设定 0.0-99999.0 mL(0.1ml)
	O_RuntimeSet         : REAL;//运行时间设定 0.1-9999s(0.1s)
    O_RunModeSet         : INT := 2;//运行模式设定；0（传输）；1（定量计算）；2（定时定量，默认模式）；
//	O_SpeedSet      	 : REAL;//速度设定 0.1-600.0 mL(rpm)	
	O_CycleNumber		 : INT;//循环次数
	O_ModuleAddress			: INT;//灌装单元地址
	O_ModuleSpeed			: REAL;//灌装单元转速
	O_ModuleStart			: INT;//灌装单元启停；1，启动；0，停止	
	O_ModuleRealVolume		: REAL;//实际灌装量	(0.1-9999.99ml)	
	O_ModuleMicroReg		: INT;//灌装量微调1,+;0-
	O_ResetCalcoeff			: INT;//恢复校准系数	
	O_BackAngle					:INT;//回吸角度设置
	I_RunSignal				:INT;//1,运行，0，停止
	I_CalSignal				:INT;//1，校准中，0，停止
END_STRUCT
END_TYPE

// ---- POUs/003_FB/53_RudongPump/08_PeristalticPumpFB/DUTs/RudongPump_Ope.TcDUT
TYPE RudongPump_Ope :
STRUCT
	xConfigure_Hmi,xConfigure_Auto 					: BOOL;
	xPush_Hmi,xPush_Auto 										: ARRAY[1..5] OF BOOL;
	xPull_Hmi,xPull_Auto 										: ARRAY[1..5] OF BOOL;	
	xStop_Hmi,xStop_Auto 										: BOOL;
	xFullSpeedPush_Hmi,xFullSpeedPush_Auto 	: BOOL;
	xFullSpeedPull_Hmi,xFullSpeedPull_Auto 	: BOOL;
	xFullSpeedStop_Hmi,xFullSpeedStop_Auto 	: BOOL;
	xPumpCal_Hmi,xPumpCal_Auto 							: BOOL;	
	xCalParWrite_Hmi,xCalParWrite_Auto 			: BOOL;
	xResetCalcoeffCal_Hmi										: BOOL;	
	
END_STRUCT
END_TYPE

// ---- POUs/003_FB/53_RudongPump/08_PeristalticPumpFB/DUTs/RudongPump_PumpHeadType.TcDUT
//保定申辰蠕动泵泵头类型选择
TYPE RudongPump_PumpHeadType :
(
	MiniPump01:=1,
	MiniPump02:=2,	
	
	HandyPump01:=3,
	HandyPump02:=4,	
	
	EasyPumpI_III:=5,//单通道
	EasyPumpII_IV:=6,//单通道
	EasyPumpV_VI:=7,//双通道

	AMC1_AMC12:=8,//适用(内径x壁厚0.13-3/0.8-1mm)
	YZ1515x:=9,//适用13#,14#,16#,17#,18#,19#,25#管
	YZ2515x:=10,//适用15#,24#管	
	
	DY15:=11,//
	DY25:=12,
	
	UD15:=13
);
END_TYPE

// ---- POUs/003_FB/53_RudongPump/08_PeristalticPumpFB/DUTs/RudongPump_PumpType.TcDUT
//保定申辰蠕动泵类型选择
TYPE RudongPump_PumpType :
(
	LabV:=1,//LabV系列
	LabF1:=2,//0.1-150rpm
	LabF3:=3,//0.1-350rpm	
	LabF4:=4,//0.1-600rpm	
	F:=5,//F系列
	M:=6,//M系列
	V:=7,//V系列
	BT_D:=8,//BT_D系列	
	PDS:=9,//PDS系列	,五位蠕动泵	
	DFPluse:=10//DFPluse系列
	
);
END_TYPE

// ---- POUs/003_FB/53_RudongPump/08_PeristalticPumpFB/DUTs/RudongPump_RunData.TcDUT
TYPE RudongPump_RunData :
STRUCT
	rPullFluVolume			:ARRAY[1..5] OF  REAL;//液量设定 0.0-99999.0 mL(0.1ml)
	rPushFluVolume			:ARRAY[1..5] OF  REAL;//液量设定 0.0-99999.0 mL(0.1ml)	
	rPullRuntime			:ARRAY[1..5] OF  REAL;//运行时间设定 0.1-9999s(0.1s)
	rPushRuntime			:ARRAY[1..5] OF  REAL;//运行时间设定 0.1-9999s(0.1s)	
	iPullBackAngle		:ARRAY[1..5] OF  INT;//回吸角度
	iPullCycleNumber		:ARRAY[1..5] OF  INT;//重复次数	
	iPushCycleNumber		:ARRAY[1..5] OF  INT;//重复次数	
	iPushBackAngle			:ARRAY[1..5] OF INT;//回吸角度
	
	iPumpType					: RudongPump_PumpType;//泵类型选择
	iPumpTypeSet				: RudongPump_PumpHeadType;//泵头类型
	iHosePipeTypeSet			: RudongPump_SoftPipeType;//软管类型	
	
	iModuleAdress		:INT;//灌装单元地址
	rModuleSpeed		:REAL;//灌装单元速度
	rModuleRealFluVolume:REAL;//实际灌装量
	rCalFluVolume		:REAL;//校准液量
	rCalTime			:REAL;//校准时间
	rCalNum				:INT;//校准加液次数	

END_STRUCT
END_TYPE

// ---- POUs/003_FB/53_RudongPump/08_PeristalticPumpFB/DUTs/RudongPump_SoftPipeType.TcDUT
//保定申辰蠕动泵软管类型选择,用前缀P表示软管,后面数字表示软管类型(内径X壁厚)
TYPE RudongPump_SoftPipeType :
(
	P13:=1,//13#软管,0.8x1.6
	P14:=2,//14#软管,1.6x1.6
	P15:=15,//15#软管,1.6x1.6
	P19:=3,//19#软管,2.4x1.6
	P16:=4,//16软管,3.1x1.6
	P25:=5,//25#软管,4.8x1.6	
	P1_1:=6,//1x1#软管,1x1
	P2_1:=7,//2x1#软管,2x1
	P2_5_1:=8,//2.5x1#软管,2.5x1	
	P3_1:=9,//3x1#软管,3x1
	P17:=10,//17#软管,6.4x1.6		
	P18:=11,//18#软管,7.9x1.6	
	P24:=12,//24#软管,6.4x2.4		
	P35:=13,//34#软管,7.9x2.4
	P36:=14//36#软管,9.6x2.4
	
	
);
END_TYPE

// ---- POUs/003_FB/53_RudongPump/08_PeristalticPumpFB/DUTs/RudongPump_Sys_Para.TcDUT
{attribute 'qualified_only'}
{attribute 'strict'}
TYPE RudongPump_Sys_Para :
STRUCT
	bySlaveID 		    : BYTE;//旋转从站号(modbus RTU)
	strSlaveIP        : STRING(15) := '127.0.0.0';//modbus子站IP地址
  	iSlavePort	      : UINT:=1031;
	xPumpRunSignal    : BOOL;//泵运行信号：true（泵处于运行状态）；false(泵处于停止状态)
	iType             : INT :=2;//1:modbus RTU;2:modbus TCP(默认)
	pRunSignal		    : POINTER TO INT;//
END_STRUCT
END_TYPE

// ---- POUs/003_FB/53_RudongPump/08_PeristalticPumpFB/DUTs/STATE_1.TcDUT

TYPE STATE_1 :
(
	DORMANT,
	EXECUTING,
	DONE,
	INERROR,
	ABORTING,
	ABORTED,
	RESETING 
);
END_TYPE

// ---- POUs/003_FB/53_RudongPump/08_PeristalticPumpFB/DUTs/ST_ModbusAddress.TcDUT
TYPE ST_ModbusAddress :
STRUCT
	
iPumpType_Address								:INT;
iHosePipeType_Address						:INT;
iFluVolumeSet_Address						:INT;
iRuntimeSet_Address							:INT;
iIntervalTime_Address						:INT;
iCycleNumber_Address						:INT;
iBackAngle_Address							:INT;
iMoveDirection_Address					:INT;
iStartStop_Address							:INT;
iFullSpeedStartStop_Address			:INT;
iModuleAddress_Address					:INT;
iModuleStartStop_Address				:INT;
iModuleRealFluVolumeSet_Address	:INT;
iRecoveryCalCoefficient_Address	:INT;
END_STRUCT
END_TYPE

// ---- POUs/003_FB/53_RudongPump/08_PeristalticPumpFB/校准程序/AutoCal_CMD.TcDUT
TYPE AutoCal_CMD :
(
 	Nodef,
	Cmd_96PumpHeadCal,//校准96个泵头
	Cmd_SpecificPumpHeadCal,	//校准指定泵头
	Cmd_ContinuesInject,//连续加液测试
	Cmd_Init	//初始化
);
END_TYPE

// ---- POUs/003_FB/53_RudongPump/08_PeristalticPumpFB/校准程序/AutoCal_ERROR.TcDUT
{attribute 'qualified_only'}
{attribute 'strict'}
TYPE AutoCal_ERROR :
(
 	No_ERROR := 0,	
  	FLT_PARA             			  	:= 1, (* 参数错误 *)
  	FLT_RudongPump             			:= 2, (* 蠕动泵出错 *) 	
  	FLT_MT_MCK204C             			:= 3, (* 秤体出错 *)
  	FLT_CmdTimeOut             			:= 4, (* 指令超时 *)			
	  FLT_AutoMode	             			:= 5 (* 不在自动模式错误 *)
							
)INT;
END_TYPE

// ---- POUs/003_FB/53_RudongPump/08_PeristalticPumpFB/校准程序/STAutoCal_ParIn.TcDUT
TYPE STAutoCal_ParIn :
STRUCT
	rDensity					:REAL:=1;//物质密度
	iPumpController		:INT;//指定控制器，指针指向
	iPumpHead					:INT;//指定泵头	
	tSteadyTime				:REAL:=3;//稳定时间                	
	xInPos						:BOOL;//蠕动泵在未知
	iContinuesInjectNum	:INT:=10;//连续加液次数
	
END_STRUCT
END_TYPE

// ---- POUs/003_FB/53_RudongPump/08_PeristalticPumpFB/校准程序/STAutoCal_ParOut.TcDUT
TYPE STAutoCal_ParOut :
STRUCT
	iCalStep								:INT;//当前流程步
	rVolume									:REAL;//体积输出
	sErrorID								:STRING;//报错内容输出
	iCurrentStep						:INT;//当前流程步
	rSteadyWeight						:REAL;//稳定重量
	rContinuesInjectWeight	:ARRAY [1..30] OF	REAL;//连续加液重量采集
END_STRUCT
END_TYPE

// ---- POUs/003_FB/53_RudongPump/08_PeristalticPumpFB/校准程序/ST_AutoCalOpe.TcDUT
TYPE ST_AutoCalOpe :
STRUCT
	x96PumpHeadCal_HMI,x96PumpHeadCal_Auto										:BOOL;//触发96泵头校准程序
	xSpecificPumpHeadCal_HMI,xSpecificPumpHeadCal_Auto				:BOOL;//触发指定泵头校准程序	
	
	xContinuesInject_HMI:BOOL;//连续加液	
	xInit_Hmi,xInit_Auto																			:BOOL;//初始化校准程序
END_STRUCT
END_TYPE

// ---- POUs/003_FB/53_RudongPump/08_PeristalticPumpFB/校准程序/ST_AutoCal_SysPar.TcDUT
TYPE ST_AutoCal_SysPar :
STRUCT
	fbMTMCK204C				: POINTER TO FB_MKC204C;//调用秤体FB
	fbRuDongPump			: POINTER TO FB_RuDongPump_modbus_DF600Plus;//调用蠕动泵FB	
	iRuDongPumpHeadNum		:INT:=9;//蠕动泵数量,最大不超过32
END_STRUCT
END_TYPE

// ---- POUs/003_FB/53_RudongPump/09_PeristalticPumpFB/RudongPump_CMD_1.TcDUT
{attribute 'qualified_only' := ''}
{attribute 'strict' := ''}
TYPE RudongPump_CMD_1 :
(
	Nodef,
	///配置指令（泵头和软管指令）
	Cmd_Configure,
	///注液指令
	Cmd_Push,
	///吸液指令 
	Cmd_Pull,
	///停止指令
	Cmd_Stop,
	///全速启动
	Cmd_FullSpeedPush,
	///全速启动
	Cmd_FullSpeedPull,
	///全速停止
	Cmd_FullSpeedStop,
	///校准泵头
	Cmd_CalPump,
	///校准泵头
	Cmd_CalReset,
	///校准参数写入
	Cmd_CalParWrite
);
END_TYPE

// ---- POUs/003_FB/53_RudongPump/09_PeristalticPumpFB/RudongPump_ERROR_1.TcDUT
{attribute 'qualified_only' := ''}
{attribute 'strict' := ''}
TYPE RudongPump_ERROR_1 :
(
	No_ERROR := 0,
	/// E-Gripper Parameter fault   程序配置参数有问题 
	FLT_PARA := 1,
	/// E-Gripper not ready 旋转有通信报警
	FLT_CONNECT := 2,
	/// E-Gripper read/write command while not ready 预留
	FLT_RDYCMD := 3,
	/// 配置参数错误 
	FLT_CONFIGURE_PARA := 4,
	/// 流量时间配置错误 
	FLT_FLUVOLUM_TIME_PARA := 5,
	/// E-Gripper release  execute Timeout 
	FLT_PUSH_TIMEOUT := 10,
	/// E-Gripper org  execute Timeout 
	FLT_PULL_TIMEOUT := 11,
	/// E-Gripper org command execute Timeout 
	FLT_STOP_TIMEOUT := 12,
	/// E-Gripper org command execute Timeout 
	FLT_FULLSPEEDSTOP_TIMEOUT := 13,
	/// E-Gripper org command execute Timeout 
	FLT_FULLSPEEDSTART_TIMEOUT := 14,
	/// E-Gripper release command execute Timeout 
	FLT_CMD_TIMEOUT := 15,
	/// E-Gripper release command execute Timeout 
	FLT_RUN_FALL := 16,
	/// E-Gripper org  execute Timeout 
	FLT_PumpCal_TIMEOUT := 17,
	/// E-Gripper org  execute Timeout 
	FLT_PumpCal_OverFlow := 18,
	/// Modbus 
	FLT_Mobdus := 19
);
END_TYPE

// ---- POUs/003_FB/53_RudongPump/09_PeristalticPumpFB/RudongPump_IOData_1.TcDUT
TYPE RudongPump_IOData_1 :
STRUCT
	///泵头型号(0-8)
	O_PumpType: INT;
	///软管型号
	O_HosePipeType: INT;
END_STRUCT
END_TYPE

// ---- POUs/003_FB/53_RudongPump/09_PeristalticPumpFB/RuDongPump_ModbusAddress.TcDUT
TYPE RuDongPump_ModbusAddress :
STRUCT
	///泵头型号设定地址
	iPumpType_Address: WORD;
	///软管型号设定地址
	iHosePipeType_Address: WORD;
	///罐装量设定地址
	iFluVolumeSet_Address: WORD;
	///罐装时间设定地址	
	iRuntimeSet_Address: WORD;
	///罐装间隔时间设定地址	
	iIntervalTime_Address: WORD;
	///罐装次数设定地址		
	iCycleNumber_Address: WORD;
	///回吸角度设定地址		
	iBackAngle_Address: WORD;
	///运行方向设定地址		
	iMoveDirection_Address: WORD;
	///启停控制设定地址		
	iStartStop_Address: WORD;
	///全速启停控制设定地址		
	iFullSpeedStartStop_Address: WORD;
	///灌装单元地址设定地址	
	iModuleAddress_Address: WORD;
	///灌装单元启停控制设定地址		
	iModuleStartStop_Address: WORD;
	///实际罐装量设定地址		
	iModuleRealFluVolumeSet_Address: WORD;
	///恢复校准系数设定地址		
	iRecoveryCalCoefficient_Address: WORD;
END_STRUCT
END_TYPE

// ---- POUs/003_FB/53_RudongPump/09_PeristalticPumpFB/RudongPump_Ope_1.TcDUT
TYPE RudongPump_Ope_1 :
STRUCT
	xConfigure_Hmi: BOOL;
	xConfigure_Auto: BOOL;
	xPush_Hmi: ARRAY[1..5] OF BOOL;
	xPush_Auto: ARRAY[1..5] OF BOOL;
	xPull_Hmi: ARRAY[1..5] OF BOOL;
	xPull_Auto: ARRAY[1..5] OF BOOL;
	xStop_Hmi: BOOL;
	xStop_Auto: BOOL;
	xFullSpeedPush_Hmi: BOOL;
	xFullSpeedPush_Auto: BOOL;
	xFullSpeedPull_Hmi: BOOL;
	xFullSpeedPull_Auto: BOOL;
	xFullSpeedStop_Hmi: BOOL;
	xFullSpeedStop_Auto: BOOL;
	xPumpCal_Hmi: BOOL;
	xPumpCal_Auto: BOOL;
	xCalParWrite_Hmi: BOOL;
	xCalParWrite_Auto: BOOL;
	xResetCalcoeffCal_Hmi: BOOL;
END_STRUCT
END_TYPE

// ---- POUs/003_FB/53_RudongPump/09_PeristalticPumpFB/RudongPump_PumpHeadType_1.TcDUT
///保定申辰蠕动泵泵头类型选择
TYPE RudongPump_PumpHeadType_1 :
(
	MiniPump01 := 1,
	MiniPump02 := 2,
	HandyPump01 := 3,
	HandyPump02 := 4,
	///单通道
	EasyPumpI_III := 5,
	///单通道
	EasyPumpII_IV := 6,
	///双通道
	EasyPumpV_VI := 7,
	///适用(内径x壁厚0.13-3/0.8-1mm)
	AMC1_AMC12 := 8,
	///适用13#,14#,16#,17#,18#,19#,25#管
	YZ1515x := 9,
	///适用15#,24#管	
	YZ2515x := 10,
	DY15 := 11,
	DY25 := 12,
	UD15 := 13
);
END_TYPE

// ---- POUs/003_FB/53_RudongPump/09_PeristalticPumpFB/RudongPump_PumpType_1.TcDUT
///保定申辰蠕动泵类型选择
TYPE RudongPump_PumpType_1 :
(
	///LabV系列
	LabV := 1,
	///0.1-150rpm
	LabF1 := 2,
	///0.1-350rpm	
	LabF3 := 3,
	///0.1-600rpm	
	LabF4 := 4,
	///F系列
	F := 5,
	///M系列
	M := 6,
	///V系列
	V := 7,
	///BT_D系列	
	BT_D := 8,
	///PDS系列	,五位蠕动泵	
	PDS := 9,
	///DFPluse系列
	DFPluse := 10
);
END_TYPE

// ---- POUs/003_FB/53_RudongPump/09_PeristalticPumpFB/RudongPump_RunData_1.TcDUT
TYPE RudongPump_RunData_1 :
STRUCT
	///液量设定 0.0-99999.0 mL(0.1ml)
	rPullFluVolume: ARRAY[1..5] OF REAL;
	///液量设定 0.0-99999.0 mL(0.1ml)	
	rPushFluVolume: ARRAY[1..5] OF REAL;
	///运行时间设定 0.1-9999s(0.1s)
	rPullRuntime: ARRAY[1..5] OF REAL;
	///运行时间设定 0.1-9999s(0.1s)	
	rPushRuntime: ARRAY[1..5] OF REAL;
	///重复次数	
	iPullCycleNumber: ARRAY[1..5] OF INT;
	///重复次数	
	iPushCycleNumber: ARRAY[1..5] OF INT;
	///泵类型选择
	iPumpType: RudongPump_PumpType;
	///泵头类型
	iPumpTypeSet: RudongPump_PumpHeadType;
	///软管类型	
	iHosePipeTypeSet: RudongPump_SoftPipeType;
	///灌装单元地址
	iModuleAdress: INT;
	///灌装单元速度
	rModuleSpeed: REAL;
	///实际灌装量
	rModuleRealFluVolume: REAL;
	///校准液量
	rCalFluVolume: REAL;
	///校准时间
	rCalTime: REAL;
	///校准加液次数	
	rCalNum: INT;

END_STRUCT
END_TYPE

// ---- POUs/003_FB/53_RudongPump/09_PeristalticPumpFB/RudongPump_SoftPipeType_1.TcDUT
///保定申辰蠕动泵软管类型选择,用前缀P表示软管,后面数字表示软管类型(内径X壁厚)
TYPE RudongPump_SoftPipeType_1 :
(
	///13#软管,0.8x1.6
	P13 := 1,
	///14#软管,1.6x1.6
	P14 := 2,
	///15#软管,1.6x1.6
	P15 := 15,
	///19#软管,2.4x1.6
	P19 := 3,
	///16软管,3.1x1.6
	P16 := 4,
	///25#软管,4.8x1.6	
	P25 := 5,
	///1x1#软管,1x1
	P1_1 := 6,
	///2x1#软管,2x1
	P2_1 := 7,
	///2.5x1#软管,2.5x1	
	P2_5_1 := 8,
	///3x1#软管,3x1
	P3_1 := 9,
	///17#软管,6.4x1.6		
	P17 := 10,
	///18#软管,7.9x1.6	
	P18 := 11,
	///24#软管,6.4x2.4		
	P24 := 12,
	///34#软管,7.9x2.4
	P35 := 13,
	///36#软管,9.6x2.4
	P36 := 14
);
END_TYPE

// ---- POUs/003_FB/53_RudongPump/09_PeristalticPumpFB/RudongPump_Sys_Para_1.TcDUT
{attribute 'qualified_only' := ''}
{attribute 'strict' := ''}
TYPE RudongPump_Sys_Para_1 :
STRUCT
	///从站号(modbus)
	bySlaveID: BYTE;
	///modbus子站IP地址	
	strSlaveIP: STRING(15) := '127.0.0.0';
	nRemotePort: INT;
END_STRUCT
END_TYPE

// ---- POUs/003_FB/53_RudongPump/41 Modbus指令/ModbusParIn.TcDUT
TYPE ModbusParIn :
STRUCT
	///数据输入	
	aSendBuffer: ARRAY[1..255] OF BYTE;
	///保持寄存器起始地址
	iHoldingRegisterAddress: WORD := 16#0;
	///保持寄存器数量	,1-125
	iHoldingRegisterNum: WORD := 16#1;
	///线圈起始地址
	iCoilStartAddress: WORD := 16#0;
	///线圈数量	,1-2000
	iCoilNum: WORD := 16#1;
END_STRUCT
END_TYPE

// ---- POUs/003_FB/53_RudongPump/41 Modbus指令/ModbusParOut.TcDUT
TYPE ModbusParOut :
STRUCT
	///寄存器字节输出
	aRcvBuffer: ARRAY[1..255] OF BYTE;
	///线圈输出		
	aRcvCoilBuffer: ARRAY[1..2000] OF BOOL;
END_STRUCT
END_TYPE

// ---- POUs/003_FB/53_RudongPump/41 Modbus指令/Modbus_Cmd.TcDUT
{attribute 'qualified_only' := ''}
{attribute 'strict' := ''}
TYPE Modbus_Cmd :
(
	Null := 0,
	///功能码01，(0X)
	ReadCoilStatus := 1,
	///功能码02，(1X)
	ReadInputStatus := 2,
	///功能码03，(4X)
	ReadHoldingRegisters := 3,
	///功能码04，(3X)
	ReadInputRegisters := 4,
	///强制单线圈05
	SetSingalCoil := 5,
	///预置单寄存器
	SetSingalHoldingRegister := 6,
	///强制多线圈
	SetMultiCoil := 15,
	///预置多寄存器			
	SetMultiHoldingRegister := 16
);
END_TYPE

// ---- POUs/003_FB/53_RudongPump/41 Modbus指令/Modbus_ErrorCode.TcDUT
{attribute 'qualified_only' := ''}
{attribute 'strict' := ''}
TYPE Modbus_ErrorCode :
(
	No_ERROR := 0,
	///无效指令
	FLT_CMD := 1,
	///指令发送错误
	FLT_SEND_ERROR := 2,
	///指令接收错误
	FLT_RECEIVE_ERROR := 3,
	///执行超时错误
	FLT_CMDTIMEOUT := 4,
	///参数溢出错误
	FLT_PAROVERFLOW := 5,
	///MODBUS错误
	FLT_MODBUS_ERROR := 6,
	///无响应
	FLT_NoResponse := 7
);
END_TYPE

// ---- POUs/003_FB/53_RudongPump/41 Modbus指令/Modbus_Operation.TcDUT
TYPE Modbus_Operation :
STRUCT
	///功能码01	
	xReadCoilStatus: BOOL;
	///功能码02					
	xReadInputStatus: BOOL;
	///功能码03
	xReadHoldingRegisters: BOOL;
	///功能码04
	xReadInputRegisters: BOOL;
	///功能码05
	xSetSingalCoil: BOOL;
	///功能码06
	xSetSingalHoldingRegister: BOOL;
	///功能码15
	xSetMultiCoil: BOOL;
	///功能码16
	xSetMultiHoldingRegister: BOOL;
END_STRUCT
END_TYPE

// ---- POUs/003_FB/53_RudongPump/41 Modbus指令/Modbus_SysPar.TcDUT
TYPE Modbus_SysPar :
STRUCT
	sRemoteHost: T_IPv4Addr;
	nRemotePort: UINT := 4008;
	///从站通信地址	
	xSlaveAdr: BYTE := 16#1;
END_STRUCT
END_TYPE

// ---- POUs/003_FB/Z_ERG_20 FB/DUTs/ERG_20_CMD.TcDUT
TYPE ERG_20_CMD :
(
  Nodef,
	Cmd_Clamp,//夹紧指令
	Cmd_Release,//松开指令
	Cmd_RotateAbsClamp,//绝对旋转夹紧指令
	Cmd_RotateAbsRelease,//绝对旋转松开指令
	Cmd_RotateRelClamp,//绝对旋转夹紧指令
	Cmd_RotateRelRelease,//绝对旋转松开指令
	Cmd_Org//初始化指令
);
END_TYPE

// ---- POUs/003_FB/Z_ERG_20 FB/DUTs/ERG_20_ERROR.TcDUT
TYPE ERG_20_ERROR :
(
	NO_ERROR := 0,	
  FLT_PARA                := 1, (* E-Gripper 参数配置有错误*)
  FLT_CONNECT             := 2, (* E-Gripper not ready 有通信报警*)
  FLT_RDYCMD              := 3, (* E-Gripper read/write command while not ready 预留*)
	FLT_DEVICE_ERROR        := 4, (*驱动器报警*)
	FLT_POWERON             := 5, (*没有上电*)
  
  FLT_CLAMP_TIMEOUT       := 10, (* E-Gripper 夹紧超时 *)
  FLT_ROTATE_TIMEOUT      := 11, (* E-Gripper 松开超时 *)
  FLT_ORG_TIMEOUT         := 12, (* E-Gripper 回原点超时 *)
	FLT_CLAMPCMD_TIMEOUT    := 13, (* E-Gripper 夹紧指令执行超时 *)
  FLT_ROTATECMD_TIMEOUT   := 14, (* E-Gripper 松开指令执行超时 *)
  FLT_ORGCMD_TIMEOUT      := 15, (* E-Gripper 回原点指令执行超时 *)
	FLT_CLAMP_DROP          := 16, (*物体掉落*)
  
  FLT_xRefOk              := 20, (* E-Gripper reference not OK 没有回原点过程中执行指令*)
	FLT_CLAMP_PARA          := 21, (* E-Gripper Clamp Para error 发送夹紧参数错误*)
	
	FLT_ClAMP_RELEASEFAIL  		       := 24, (* E-Gripper 松开指令超时*)
  FLT_ClAMP_CLAMPFAIL        	     := 25, (* E-Gripper 夹紧物体失败 *)
	FLT_ROTATE_CLAMPFAIL        	   := 26, (* E-Gripper 关盖失败*)
	FLT_ROTATE_RELEASEFAIL  		     := 27 (* E-Gripper 开盖失败 *)	
)INT;
END_TYPE

// ---- POUs/003_FB/Z_ERG_20 FB/DUTs/ST_ERG_20_IOData.TcDUT
TYPE ST_ERG_20_IOData ://IO数据
STRUCT
	//夹持输入数据映射
	I_ClampInit        : INT;//夹持初始化状态：0：夹持未初始化；5：夹持初始化成功  其它：初始化中
	I_ClampState       : INT;//0：运动到位，1：到达中；2：夹住物体；3：物体掉落
	I_ClampCurrentPos       : REAL;//反馈当前夹爪实时位置  0-30mm(目标位置偏差0.02)
	I_ClampCurrentSpeed     : REAL;//反馈当前夹爪实时速度  (1-200mm)	
	I_ClampCurrentForce     : REAL;//反馈当前夹爪实时力值b ( 0.2 - 0.5A ) 
	//旋转输入数据映射
	I_RotateState       : INT;//0：到位，1，运动中，2：堵转
	I_RotateCurrentPos       : REAL;//单位 mm
	I_RotateCurrentSpeed     : REAL;//单位 mm/s
	I_RotateCurrentForce     : REAL;//单位 A
	I_DeviceERRORState : INT;//保留中（供应商暂时没有提供功能）
	//输出数据映射
	O_Init : INT;//写入 1：回零位（找单向位置） 
  //夹持数据设置 
	O_ClampForceSet : REAL;//设置力值( 0.1 - 0.5A ) 走位置时将扭矩设置最小设置成0.3
	O_ClampPosSet : REAL;//设定夹爪位置( 0-20mm)
	O_ClampSpeedSet : REAL;//以设定速度运行(1-400mm)	
	//旋转数据设置
	O_RotateForceSet : REAL;//设置力值( 0.2~1A )    最小值设置成0.3
	O_RotatePosSet : REAL;//设定夹爪旋转角度( -3600000~360000 度)
	O_RotateSpeedSet : REAL;//以设定速度运行(取值范围：1~1440度/秒)	
END_STRUCT
END_TYPE

// ---- POUs/003_FB/Z_ERG_20 FB/DUTs/ST_ERG_20_Sys_Para.TcDUT
TYPE ST_ERG_20_Sys_Para :
STRUCT	
  //pOutputData       : POINTER TO INT;//0:回原点控制数据;1-2:夹持位置设置;3-4:夹持速度设置;5-6:夹持电流设置;7-8:夹持位置设置;11-12:夹持速度设置;13-14:夹持电流设置
	//pInputData   		  : POINTER TO INT;//0:初始化状态反馈;1:夹持状态反馈;2-3:夹持位置反馈;4-5:夹持速度反馈;6-7:夹持电流反馈 8:旋转状态 10-11:旋转角度反馈:12-13:旋转速度反馈;14-15:旋转电流反馈 16-17:报警信息
	///modbus子站IP地址
	strSlaveIP: STRING(15) := '127.0.0.0';
	///默认是502
	iSlavePort: UINT := 502;
	///modbus rtu子站地址	
	bySlaveID: BYTE;
END_STRUCT
END_TYPE

// ---- POUs/003_FB/Z_ERG_20 FB/DUTs/ST_Huiling_Pers_Para.TcDUT
TYPE ST_Huiling_Pers_Para :
STRUCT
	aHMIClampPara , aHMIReleasePara : ARRAY[1..5] OF ST_Huiling_PosPara;//夹紧轴点位信息
	aHMIRotateClampPara , aHMIRotateReleasePara : ARRAY[1..5] OF ST_Huiling_PosPara;//旋转轴点位信息
	aHMIRotateRelClampPara , aHMIRotateRelReleasePara : ARRAY[1..5] OF ST_Huiling_PosPara;//旋转轴点位信息
END_STRUCT
END_TYPE

// ---- POUs/003_FB/Z_ERG_20 FB/DUTs/ST_Huiling_PosPara.TcDUT
TYPE ST_Huiling_PosPara :
STRUCT
	rTorqueSet   : REAL;//目标力值设置  ( 0.2 - 0.5A )
	rSpeedSet    : REAL;//运行速度设置  (1-200mm)	
	rPosAngleSet : REAL;//位置和速度设置值	 ( 0-30mm)
END_STRUCT
END_TYPE

// ---- POUs/40_TcpIp/40_TcpIp/E_ClientSteps.TcDUT
{attribute 'tc_no_symbol'}
TYPE E_ClientSteps :
(
	CLIENT_STATE_IDLE,//空闲状态
	CLIENT_STATE_CONNECT_START,//启动网络连接
	CLIENT_STATE_CONNECT_WAIT,//等待连接完成
	CLIENT_STATE_DATAEXCHA_START,//启动数据收发操作
	CLIENT_STATE_DATAEXCHA_WAIT,//等待数据收发完成
	CLIENT_STATE_CLOSE_START,//启动关闭连接操作
	CLIENT_STATE_CLOSE_WAIT,//等待关闭完成
	
//	CLIENT_STATE_IDLE,
//	CLIENT_STATE_CONNECT_START,
//	CLIENT_STATE_CONNECT_WAIT,
	CLIENT_STATE_SEND_START,
	CLIENT_STATE_SEND_WAIT,
	CLIENT_STATE_WAITTIME1,
	CLIENT_STATE_WAITTIME2,
	CLIENT_STATE_RECIVE_START,
	CLIENT_STATE_RECIVE_WAIT,
	//CLIENT_STATE_CLOSE_START,
	//CLIENT_STATE_CLOSE_WAIT,
	CLIENT_STATE_ERROR,
	CLIENT_STATE_DONE
	
	
	
	
);
END_TYPE

// ---- GVLs/Common.TcGVL
VAR_GLOBAL 
	
   //工站清料完成信号
    abClearMaterialOver  : ARRAY [1..16] OF BOOL;//
   //工站产品状态
	arMainlineFixtureData :  ARRAY [1..gc_MainLineFixtureNumber] OF DUT_MainlineFixture;
	arBeltLineFixtureData	:	ARRAY[1..gc_BeltLineFixtureNumber] OF DUT_BeltLineFixture;
	
	arRobot2ProductStatus :  DUT_Robot2;
 	arMainLineFixturePos 	 		: ARRAY [0..50] OF REAL;
	
	_MainlineFristRun: BOOL;
	_wRefCounter: WORD;
	_FirstSetValue: BOOL;
	
END_VAR
VAR_GLOBAL CONSTANT

END_VAR


VAR_GLOBAL PERSISTENT
		arCurFixtureNumStation		 	 : ARRAY[1..20] OF  DINT;
END_VAR

// ---- GVLs/GVL_Config.TcGVL
VAR_GLOBAL CONSTANT
	gc_xEstopYesORno               		  : BOOL:=1;   //机器拍急停:1-停机重新初始化，0-继续跑不用初始化
	gc_uiAxisNum						  : INT:=19;//轴数量
	gc_uiAxisMoveNum          			 : INT:=10 ;  //轴点位数量
	gc_uiCylinderNum					  : INT:=50; //气缸数量 
	gc_uiMachineNum						 : INT:=1;	//机器数量
	gc_uiStationNum				 		  : INT:=16;//工站数量
	gc_uiHMI_Num						  : INT:=2;	//人机界面数量
	gc_uiPXF5Num							 :INT:=2;//温控器个数
	gc_uiRGI_14_Number                	 	: INT :=1 ;  //大寰电动夹爪（旋转+夹紧）
	gc_uiHITBOT_Number						: INT :=2;//惠灵电动夹爪(旋转+夹持）
	gc_uiTURINRobot_Num             	    : INT :=1 ;   //图灵机械手
	gc_uiCameraNum							: INT:= 18;//相机个数
	gc_uiRudongPump							:INT := 12;//蠕动泵控制器个数
	gc_MainLineFixtureNumber				:INT:=43;//主流线的位置数
	gc_BeltLineFixtureNumber				:INT:=6;//皮带线的位置数
	gc_MainLineAxisPositionOffset			:REAL:=36;//主流线位置偏移
	gc_StepHistory							:INT:=500;//step log数量
	gc_RecipeNum							:WORD:=1;//保存配方数量
	gc_ModuleProNo							:INT:=10;//过程数据数组大小
	gc_AliveNum									:INT:=10;//心跳包数量
	gc_uiValveNum								:INT:=2;//真空发生器个数
	gc_uiSlaveNum								:INT:=4;//电柜EtherCAT状态
	gc_uiLoadcellNum						:INT:=6;//压力传感器个数
	gc_uiCimcorNum							:INT:=1;//离子风棒个数
END_VAR

// ---- GVLs/GVL_Robot.TcGVL
VAR_GLOBAL 
	stToRobot1	: DUT_SysToRobot1; //
	stFromRobot1  : DUT_SysFromRobot1; //
END_VAR

// ---- GVLs/GVL_PC.TcGVL
VAR_GLOBAL 
  sPLC_TO_PC   			AT%MW300  :DUT_PCReceive;
  sPLC_From_PC  		AT%MW500    :DUT_PCSend;
  sCamera_TO_Plc 		AT%MW100  :DUT_CameraSend;
	sCamera_From_Plc	AT%MW150	:DUT_CameraReceive;
  sModbus_200SMART :DUT_200SMART;
END_VAR

// ---- GVLs/GVL_Standard.TcGVL
VAR_GLOBAL
	Axis						  : ARRAY[1..gc_uiAxisNum] OF AXIS_REF;
	fbAxis						: ARRAY[1..gc_uiAxisNum] 			OF FB_Axis;
	fbAxisHome						: ARRAY[1..gc_uiAxisNum] 			OF FB_AxisHome;
	fbCylinder					: ARRAY[1..gc_uiCylinderNum] 		OF FB_Cylinder;
	fbProface						: ARRAY[1..gc_uiHMI_Num] 			OF FB_Proface;
	fbMachine					: ARRAY[1..gc_uiMachineNum] 		OF FB_Machine;
	fbStation					: ARRAY[1..gc_uiStationNum] 		OF FB_Station;
	fbRGI_14_Modbus 			: ARRAY[1..gc_uiRGI_14_Number] OF FB_RGI_14_Modbus;
	fbTempretureControl           : ARRAY [1..gc_uiPXF5Num] OF FB_TempControl_FUSHI;    //modbus tcp
	fbMCK204W					  : FB_MT_MKC;//秤
	fbAutoCal					  :	FB_AutoCal;
	fbRudongPump 				:ARRAY[1..gc_uiRudongPump] OF FB_RuDongPump_modbus_DF600Plus;	
	fbTURINContorl                : ARRAY[1..gc_uiTURINRobot_Num]     OF FB_TURINContorl;
	(*fb_CommWithPC				:FB_CommWithPC;*)
	fbRecipes					:ARRAY[1..gc_RecipeNum]OF FB_Recipes;
	fbERG_20_Modbus				:ARRAY[1..gc_uiHITBOT_Number] OF FB_ERG_20_Modbus;
	fbGetTime					:FB_GetTime;
	fbCamera					:ARRAY[1..gc_uiCameraNum] OF FB_Camera;
	fbRudongPumpModbusTcp		:ARRAY[1..gc_uiRudongPump] OF FB_RuDongPump_ModbusTCP;
	fbAlive					 :ARRAY[1..gc_AliveNum] OF FB_Alive;
	fbEhterCATSlaveMonitor	:ARRAY[1..gc_uiSlaveNum] OF FB_EtherCatSlaveMonitor;
	fbModbus_200Smart				:FB_Modbus_200Smart;
	fbEncoder								:FB_Encoder;
	fbATV12									:FB_ATV12;
	fbMCK										 :FB_MKC204C;
	fbERG										 :ARRAY[1..gc_uiHITBOT_Number] OF FB_ERG_20C;
	fbSmcVacuum							:ARRAY[1..gc_uiValveNum] OF FB_SmcVacuum;
	fbLoadCell							:ARRAY[1..gc_uiLoadcellNum] OF FB_LoadCell;
	fbCimcor								:ARRAY[1..gc_uiCimcorNum] OF FB_Cimcor_IZN10E;
	fbEasyPumps							:ARRAY[1..gc_uiRudongPump] OF FB_KF300;
   xNot_power					: ARRAY[1..gc_uiAxisNum] OF BOOL;//设原点时断使能
	cnSlaveAddr	        : ARRAY[1..gc_uiAxisNum] OF UINT;//伺服的从站地址
	sDeviceNetId AT%I* : AmsNetID ; //设备的ethercat地址
	sEctNetId : STRING ;//需要将读到的地址转成string

	home_method : ARRAY[1..gc_uiAxisNum] OF SINT := [gc_uiAxisNum(35)];	
	bSetPosDone	: ARRAY[1..gc_uiAxisNum] OF BOOL;
	(*其他信号*)
	strDoorBypassHmi	:BOOL;
	xMachineLamp		:BOOL;
	xultravioletLampControl:BOOL;///紫外灯控制按钮
	xultravioletButtonLamp	:BOOL;
	
	strLocalDateTime: STRING;
	
	xMainLineRunTestHMI:BOOL;//环形线运行测试按钮
	
	axBypassSignal	:ARRAY[1..50] OF BOOL ;//[1]-上料工位相机屏蔽  //[2]-注液屏蔽  [3]-相机液位检测屏蔽  [4]-热封铝膜屏蔽
	//
	stPara: INT;
	aReleaseControl: INT;
	arFlowLineControl  :  ARRAY[1..2] OF BOOL; //[1]-启动   [2]-停止
	arAxisSensor	 AT%I*:ARRAY[1..gc_uiAxisNum] OF UDINT;
	
	arAxisSensorN:ARRAY[1..gc_uiAxisNum] OF BOOL;//负极限
	arAxisSensorP:ARRAY[1..gc_uiAxisNum] OF BOOL;//正极限
	arAxisSensorH:ARRAY[1..gc_uiAxisNum] OF BOOL;//原点
	
	xS05WorkPermit : BOOL;//切莫工位允许调整工位动作
	
	xAllRudongPumpEmpty:BOOL;//所有蠕动泵排空
	xRudongPumpEmptyDone:BOOL;//排空结束
	arxRudongPumpEmptyBypass:ARRAY[1..12] OF BOOL;//蠕动泵排空屏蔽	
	arxRudongPumpCalibBypass:ARRAY[1..12] OF BOOL;//蠕动泵校准功能屏蔽	
	stManualCalib:stEasyPumpsParamter;//手动校准功能
END_VAR

VAR_GLOBAL 
	stToRobot,stToRobotZero       : DUT_SysToRobot; //
	stFromRobot,stFromRobotZero   : DUT_SysFromRobot; //
	// 深孔板选择
	iBoxChoose: INT:=1;
	//允许主流线运行
	xS07MainlineRunPermit	:BOOL;
	//程序编号调用
	asModuleSeqData	    	:ARRAY[1..gc_uiStationNum] OF tsPartSequence;(*module sequence *)
	stZ_ERG_20_IOData      :ARRAY[1..gc_uiHITBOT_Number] OF ST_ERG_20_IOData;
	//相机检测工位检测结果
	arCameraResultHmi:ARRAY[1..5,1..4,1..12] OF INT;
	//相机结果中转
	arCameraResult:ARRAY[1..gc_uiCameraNum] OF INT;
	//各工位手动NG触摸屏按钮
	arManualNOKHmiButton:ARRAY[1..gc_uiStationNum] OF  BOOL;
	//屏蔽蜂鸣器
	_BuzzerBypassButton:BOOL;
	_BuzzerBypassLamp:BOOL;
	//相机检测工位循环选择
	bS03Counter:BYTE:=1;
	//铝膜吹气电磁阀
	xS06AluBlowValve:BOOL;
END_VAR

VAR_GLOBAL PERSISTENT
	stData	 					:ST_Recipe;
	arStepAuto					:DUT_Sta;
	arStepInit					:DUT_Sta;
	stCalibration			:DUT_Calibration;
END_VAR

// ---- GVLs/GVL_System.TcGVL

VAR_GLOBAL CONSTANT
	bOn							: BOOL:=TRUE;			//常On
	bOff						: BOOL:=FALSE;			//常Off
	rPai						: LREAL:=3.14159265358979323846264338327950238;
END_VAR

VAR_GLOBAL
	stSysPulse         : ST_SysPulse ;
END_VAR

// ---- GVLs/GVL_UPS.TcGVL
{attribute 'qualified_only'}
VAR_GLOBAL
	fb_1sUPS						: FB_S_UPS_CX51x0;///用于配有1sUPS的PLC
END_VAR

// ---- GVLs/IO.TcGVL
VAR_GLOBAL 
//电柜+ET01
    ET01_Input AT %I* : ARRAY [1..6] OF EL1889;//输入
    ET01_Output AT %Q* : ARRAY [1..6] OF EL2889;//输出
	
		ET02_Input AT %I* : ARRAY [1..6] OF EL1889;//输入
    ET02_Output AT %Q* : ARRAY [1..5] OF EL2889;//输出
	
		ET03_Input AT %I* : ARRAY [1..1] OF EL1889;//输入
		ET03_Output AT %Q* : ARRAY [1..1] OF EL2889;//输出
	
		ET04_Input AT %I* : ARRAY [1..2] OF EL1889;//输入
    ET04_Output AT %Q* : ARRAY [1..2] OF EL2889;//输出
	
	arEtherCATWcState AT %I* : ARRAY [1..20] OF BOOL;//输出
	uiStatusCopy		AT %I*   : ARRAY[1..gc_uiAxisNum] OF  USINT;
IxSafetyRelayOK	:BOOL;//	安全继电器信号
IxStartButton	:BOOL;//	启动按钮信号
IxStopButton	:BOOL;//	停止按钮信号
IxResetButton	:BOOL;//	复位按钮信号
IxInitButton	:BOOL;//	初始化按钮信号
IxAutoMode	:BOOL;//	自动模式信号
IxManualMode	:BOOL;//	手动模式信号
IxAirPressure	:BOOL;//	上料工位¶气压检测
IxS01PositionSensor1	:BOOL;//	链板线深孔板¶位置1传感器
IxS01PositionSensor2	:BOOL;//	链板线深孔板¶位置2传感器
IxS01PositionSensor3	:BOOL;//	链板线深孔板¶位置3传感器
IxS01PositionSensor4	:BOOL;//	链板线深孔板¶位置4传感器
IxS01Sensor1Reached	:BOOL;//	上料工位¶到位传感器1
IxS01Sensor2Reached	:BOOL;//	上料工位¶到位传感器2
IxS02Sensor1Reached	:BOOL;//	注液工位¶到位传感器1
IxS02Sensor2Reached	:BOOL;//	注液工位¶到位传感器2
Ixshare2	:BOOL;//	备用1
Ixshare3	:BOOL;//	备用2
Ixshare4	:BOOL;//	备用3
Ixshare5	:BOOL;//	备用4
IxS03Sensor1Reached	:BOOL;//	相机工位¶到位传感器1
IxS03Sensor2Reached	:BOOL;//	相机工位¶到位传感器2
IxS03Sensor3Reached	:BOOL;//	相机工位¶到位传感器3
IxS03Sensor4Reached	:BOOL;//	相机工位¶到位传感器4
IxS03Sensor5Reached	:BOOL;//	相机工位¶到位传感器5
IxVFDErrorSignal	:BOOL;//	上料链板线变频器异常
Ixshare31	:BOOL;//	备用1
Ixshare32	:BOOL;//	备用2
Ixshare33	:BOOL;//	备用3
Ixshare34	:BOOL;//	备用4
IxS01SafetyDoorReady	:BOOL;//	上料工位安全门
IxS02SafetyDoorReady_2	:BOOL;//	注液工位安全门
IxS01VTCPressCyl_1WP	:BOOL;//	Z轴阻挡气缸1¶动点
IxS01VTCPressCyl_1HP	:BOOL;//	Z轴阻挡气缸1¶原点
IxS01VTCPressCyl_2WP	:BOOL;//	Z轴阻挡气缸2¶动点
IxS01VTCPressCyl_2HP	:BOOL;//	Z轴阻挡气缸2¶原点
IxS01VTCPressCyl_3WP	:BOOL;//	Z轴阻挡气缸3¶动点
IxS01VTCPressCyl_3HP	:BOOL;//	Z轴阻挡气缸3¶原点
IxS01VTCPressCyl_4WP	:BOOL;//	Z轴阻挡气缸4¶原点
IxS01VTCPressCyl_4HP	:BOOL;//	Z轴阻挡气缸4¶原点
IxS01VTCCyl_1WP	:BOOL;//	上料工位¶移栽Z轴气缸1¶动点1¶动点
IxS01VTCCyl_2WP	:BOOL;//	上料工位¶移移栽Z轴气缸
IxS01VTCCyl_1HP	:BOOL;//	上料工位¶移移栽Z轴气缸2¶动点
IxS01VTCCyl_2HP	:BOOL;//	上料工位¶移移栽Z轴气缸2¶原点
IxS02HOZAdjustCyl_1WP	:BOOL;//	注液工位¶上层水平调整气缸1¶动点
IxS02HOZAdjustCyl_1HP	:BOOL;//	注液工位¶上层水平调整气缸1¶原点
IxS02HOZAdjustCyl_2WP	:BOOL;//	注液工位¶上层水平调整气缸2¶动点
IxS02HOZAdjustCyl_2HP	:BOOL;//	注液工位¶上层水平调整气缸2¶原点
IxS02HOZAdjustCyl_3WP	:BOOL;//	注液工位¶下层水平调整气缸1¶动点
IxS02HOZAdjustCyl_3HP	:BOOL;//	注液工位¶下层水平调整气缸1¶原点点
IxS02HOZAdjustCyl_4WP	:BOOL;//	注液工位¶下层水平调整气缸2¶动点
IxS02HOZAdjustCyl_4HP	:BOOL;//	注液工位¶下层水平调整气缸2¶原点
IxS02ROTCylWP	:BOOL;//	注液工位¶防滴液气缸¶动点
IxS02ROTCylHP	:BOOL;//	注液工位¶防滴液气缸¶原点
Ixshare6	:BOOL;//	备用
Ixshare7	:BOOL;//	备用
IxS03HOZAdjustCyl_1WP	:BOOL;//	相机检测工位¶上层水平调整气缸1¶动点
IxS03HOZAdjustCyl_1HP	:BOOL;//	相机检测工位¶上层水平调整气缸1¶原点
IxS03HOZAdjustCyl_2WP	:BOOL;//	相机检测工位¶上层水平调整气缸2¶动点
IxS03HOZAdjustCyl_2HP	:BOOL;//	相机检测工位¶上层水平调整气缸2¶原点
IxS03HOZAdjustCyl_3WP	:BOOL;//	相机检测工位¶上层水平调整气缸3¶动点
IxS03HOZAdjustCyl_3HP	:BOOL;//	相机检测工位¶上层水平调整气缸3¶原点
IxS03HOZAdjustCyl_4WP	:BOOL;//	相机检测工位¶上层水平调整气缸4¶动点
IxS03HOZAdjustCyl_4HP	:BOOL;//	相机检测工位¶上层水平调整气缸4¶动点
IxS03HOZAdjustCyl_5WP	:BOOL;//	相机检测工位¶下层水平调整气缸1¶动点
IxS03HOZAdjustCyl_5HP	:BOOL;//	相机检测工位¶下层水平调整气缸1¶原点
IxS03HOZAdjustCyl_6WP	:BOOL;//	相机检测工位¶下层水平调整气缸2¶动点
IxS03HOZAdjustCyl_6HP	:BOOL;//	相机检测工位¶下层水平调整气缸2¶原点
IxS03HOZAdjustCyl_7WP	:BOOL;//	相机检测工位¶下层水平调整气缸3¶动点
IxS03HOZAdjustCyl_7HP	:BOOL;//	相机检测工位¶下层水平调整气缸3¶原点
IxS03HOZAdjustCyl_8WP	:BOOL;//	相机检测工位¶下层水平调整气缸4¶动点
IxS03HOZAdjustCyl_8HP	:BOOL;//	相机检测工位¶下层水平调整气缸4¶原点
IxErrorSignal	:BOOL;//	上料工位¶离子风棒¶异常信号
IxMaintenanceSignal	:BOOL;//	上料工位¶离子风棒¶维护信号
Ixshare9	:BOOL;//	备用
Ixshare10	:BOOL;//	备用
Ixshare11	:BOOL;//	备用
Ixshare12	:BOOL;//	备用
Ixshare13	:BOOL;//	备用
Ixshare14	:BOOL;//	备用
Ixshare15	:BOOL;//	备用
Ixshare16	:BOOL;//	备用
Ixshare17	:BOOL;//	备用
Ixshare18	:BOOL;//	备用
Ixshare19	:BOOL;//	备用
Ixshare20	:BOOL;//	备用
Ixshare21	:BOOL;//	备用
Ixshare22	:BOOL;//	备用
Ixshare23	:BOOL;//	备用
Ixshare24	:BOOL;//	备用
Ixshare25	:BOOL;//	备用
Ixshare26	:BOOL;//	备用
Ixshare27	:BOOL;//	备用
Ixshare28	:BOOL;//	备用
Ixshare29	:BOOL;//	备用
Ixshare30	:BOOL;//	备用

QxStartButtonLamp	:BOOL;//	启动按钮指示灯
QxStopButtonLamp	:BOOL;//	停止按钮指示灯
QxResetButtonLamp	:BOOL;//	复位按钮指示灯
QxInitButtonLamp	:BOOL;//	初始化按钮指示灯
QxIonStopControl	:BOOL;//	上料工位¶离子风棒¶停止放电信号
QxIonCheckDirtyControl	:BOOL;//	上料工位¶离子风棒¶电极针脏污检出信号
QxFlowLineStart	:BOOL;//	链板线电机¶正转输出
QxFlowLineStop	:BOOL;//	链板线电机¶停止输出
QxFlowLineSpeedCtrl_1	:BOOL;//	链板线电机¶多段速1输出
QxFlowLineSpeedCtrl_2	:BOOL;//	链板线电机¶多段速2输出
QxMachineLamp1Control	:BOOL;//	日光灯1控制
QxMachineLamp2Control	:BOOL;//	日光灯2控制
QxRedLamp	:BOOL;//	三色灯-红灯
QxYellowLamp	:BOOL;//	三色灯-黄灯
QxGreenLamp	:BOOL;//	三色灯-绿灯
QxBuzzer	:BOOL;//	三色-蜂鸣器灯
QxS01VTCPressCyl_1WP	:BOOL;//	链板线¶Z轴阻挡气缸1¶动点输出
QxS01VTCPressCyl_1HP	:BOOL;//	链板线¶Z轴阻挡气缸1¶原点输出
QxS01VTCPressCyl_2WP	:BOOL;//	链板线¶Z轴阻挡气缸2¶动点输出
QxS01VTCPressCyl_2HP	:BOOL;//	链板线¶Z轴阻挡气缸2¶原点输出
QxS01VTCPressCyl_3WP	:BOOL;//	链板线¶Z轴阻挡气缸3¶动点输出
QxS01VTCPressCyl_3HP	:BOOL;//	链板线¶Z轴阻挡气缸3¶原点输出
QxS01VTCPressCyl_4WP	:BOOL;//	链板线¶Z轴阻挡气缸4¶动点输出
QxS01VTCPressCyl_4HP	:BOOL;//	链板线¶Z轴阻挡气缸4¶原点输出
QxS01VTCCyl_1WP	:BOOL;//	上料工位¶移栽Z轴气缸1¶动点输出
QxS01VTCCyl_1HP	:BOOL;//	上料工位¶移栽Z轴气缸¶原点输出
QxS01VTCCyl_2WP	:BOOL;//	上料工位¶移栽Z轴气缸2¶动点输出
QxS01VTCCyl_2HP	:BOOL;//	上料工位¶移栽变距气缸¶原点输出
QxS02HOZAdjustCyl_1WP	:BOOL;//	注液工位¶上层水平调整气缸1¶动点输出
QxS02HOZAdjustCyl_1HP	:BOOL;//	注液工位¶上层水平调整气缸1¶原点输出
QxShare40	:BOOL;//	备用
QxShare41	:BOOL;//	备用
QxS02HOZAdjustCyl_3WP	:BOOL;//	注液工位¶下层水平调整气缸1¶动点输出
QxS02HOZAdjustCyl_3HP	:BOOL;//	注液工位¶下层水平调整气缸1¶原点输出
QxShare42	:BOOL;//	备用
QxShare43	:BOOL;//	备用
QxS02ROTCylWP	:BOOL;//	注液工位¶防滴液¶动点输出
QxS02ROTCylHP	:BOOL;//	注液工位¶防滴液¶原点输出
QxS03HOZAdjustCyl_1WP	:BOOL;//	相机工位¶上层水平调整气缸1¶动点输出
QxS03HOZAdjustCyl_1HP	:BOOL;//	相机工位¶上层水平调整气缸1¶原点输出
QxS03HOZAdjustCyl_2WP	:BOOL;//	相机工位¶上层水平调整气缸2¶动点输出
QxS03HOZAdjustCyl_2HP	:BOOL;//	相机工位¶上层水平调整气缸2¶原点输出
QxS03HOZAdjustCyl_3WP	:BOOL;//	相机工位¶上层水平调整气缸3¶动点输出
QxS03HOZAdjustCyl_3HP	:BOOL;//	相机工位¶上层水平调整气缸3¶原点输出
QxS03HOZAdjustCyl_4WP	:BOOL;//	相机工位¶上层水平调整气缸4¶动点输出
QxS03HOZAdjustCyl_4HP	:BOOL;//	相机工位¶上层水平调整气缸4¶原点输出
QxS03HOZAdjustCyl_5WP	:BOOL;//	相机工位¶上层水平调整气缸5¶动点输出
QxS03HOZAdjustCyl_5HP	:BOOL;//	相机工位¶上层水平调整气缸5¶原点输出
QxS03HOZAdjustCyl_6WP	:BOOL;//	相机工位¶上层水平调整气缸6¶动点输出
QxS03HOZAdjustCyl_6HP	:BOOL;//	相机工位¶上层水平调整气缸6¶原点输出
QxS03HOZAdjustCyl_7WP	:BOOL;//	相机工位¶上层水平调整气缸7¶动点输出
QxS03HOZAdjustCyl_7HP	:BOOL;//	相机工位¶上层水平调整气缸7¶原点输出
QxS03HOZAdjustCyl_8WP	:BOOL;//	相机工位¶上层水平调整气缸8¶动点输出
QxS03HOZAdjustCyl_8HP	:BOOL;//	相机工位¶上层水平调整气缸8¶原点输出
QxS04AluCoverCylWP	:BOOL;//	铝膜胀气轴气缸动点
QxShare8	:BOOL;//	备用
QxShare9	:BOOL;//	备用
QxShare10	:BOOL;//	备用
QxShare11	:BOOL;//	备用
QxShare12	:BOOL;//	备用
QxShare13	:BOOL;//	备用
QxShare14	:BOOL;//	备用
QxShare15	:BOOL;//	备用
QxShare16	:BOOL;//	备用
QxCamera1Trigger	:BOOL;//	相机检测工位¶相机触发1
QxCamera2Trigger	:BOOL;//	相机检测工位¶相机触发2
QxCamera3Trigger	:BOOL;//	相机检测工位¶相机触发3
QxCamera4Trigger	:BOOL;//	相机检测工位¶相机触发4
QxCamera5Trigger	:BOOL;//	相机检测工位¶相机触发5
QxCamera6Trigger	:BOOL;//	相机检测工位¶相机触发6
QxCamera7Trigger	:BOOL;//	相机检测工位¶相机触发7
QxCamera8Trigger	:BOOL;//	相机检测工位¶相机触发8
QxCamera9Trigger	:BOOL;//	相机检测工位¶相机触发9
QxCamera10Trigger	:BOOL;//	相机检测工位¶相机触发10
QxCamera11Trigger	:BOOL;//	相机检测工位¶相机触发11
QxCamera12Trigger	:BOOL;//	相机检测工位¶相机触发12
QxCamera13Trigger	:BOOL;//	相机检测工位¶相机触发13
QxCamera14Trigger	:BOOL;//	相机检测工位¶相机触发14
QxCamera15Trigger	:BOOL;//	相机检测工位¶相机触发15
QxCamera16Trigger	:BOOL;//	相机检测工位¶相机触发16
QxCamera17Trigger	:BOOL;//	相机检测工位¶相机触发17
QxCameraLight1Trigger	:BOOL;//	相机光源触发通道1
QxCameraLight2Trigger	:BOOL;//	相机光源触发通道2
QxCameraLight3Trigger	:BOOL;//	相机光源触发通道3
QxCameraLight4Trigger	:BOOL;//	相机光源触发通道4
QxShare21	:BOOL;//	备用
QxShare22	:BOOL;//	备用
QxShare23	:BOOL;//	备用
QxShare24	:BOOL;//	备用
QxShare25	:BOOL;//	备用
QxShare26	:BOOL;//	备用
QxShare27	:BOOL;//	备用
QxShare28	:BOOL;//	备用
QxShare29	:BOOL;//	备用
QxShare30	:BOOL;//	备用
QxShare31	:BOOL;//	备用
IxS04HOZAdjustCyl_1WP	:BOOL;//	热熔工位¶上层水平调整气缸1¶动点
IxS04HOZAdjustCyl_1HP	:BOOL;//	热熔工位¶上层水平调整气缸1¶原点
IxS04HOZAdjustCyl_2WP	:BOOL;//	热熔工位¶上层水平调整气缸2¶动点
IxS04HOZAdjustCyl_2HP	:BOOL;//	热熔工位¶上层水平调整气缸2¶原点
IxS04HOZAdjustCyl_3WP	:BOOL;//	热熔工位¶下层水平调整气缸1¶动点
IxS04HOZAdjustCyl_3HP	:BOOL;//	热熔工位¶下层水平调整气缸1¶原点
IxS04HOZAdjustCyl_4WP	:BOOL;//	热熔工位¶下层水平调整气缸2¶动点
IxS04HOZAdjustCyl_4HP	:BOOL;//	热熔+A9工位¶下层水平调整气缸2¶原点
IxS06GlampCyl_1WP	:BOOL;//	切膜工位¶前侧夹膜气缸1¶动点
IxS06GlampCyl_1HP	:BOOL;//	切膜工位¶前侧夹膜气缸1¶原点
IxS06GlampCyl_2WP	:BOOL;//	切膜工位¶前侧夹膜气缸2¶动点
IxS06GlampCyl_2HP	:BOOL;//	切膜工位¶前侧夹膜气缸2¶原点
IxS06GlampCyl_3WP	:BOOL;//	切膜工位¶后侧夹膜气缸1¶动点
IxS06GlampCyl_3HP	:BOOL;//	切膜工位¶后侧夹膜气缸1¶原点
IxS06GlampCyl_4WP	:BOOL;//	切膜工位¶后侧夹膜气缸2¶动点
IxS06GlampCyl_4HP	:BOOL;//	切膜工位¶后侧夹膜气缸2¶原点
IxS06HOZReachedCyl_1WP	:BOOL;//	切膜工位¶水平到位气缸1¶动点
IxS06HOZReachedCyl_1HP	:BOOL;//	切膜工位¶水平到位气缸1¶原点
IxS06HOZReachedCyl_2WP	:BOOL;//	切膜工位¶水平到位气缸2¶动点
IxS06HOZReachedCyl_2HP	:BOOL;//	切膜工位¶水平到位气缸2¶原点
IxS06HOZCyl_1WP	:BOOL;//	切膜工位¶水平切膜气缸¶动点
IxS06HOZCyl_1HP	:BOOL;//	切膜工位¶水平切膜气缸¶原点
IxShare60	:BOOL;//	备用
IxShare61	:BOOL;//	备用
IxS06VTCAdjustCylWP	:BOOL;//	切膜工位¶下方对中顶升气缸¶动点
IxS06VTCAdjustCylHP	:BOOL;//	切膜工位¶下方对中顶升气缸¶原点
IxS06GlampAdjustCyl_1WP	:BOOL;//	切膜工位¶下方对中夹爪气缸1¶动点
IxS06GlampAdjustCyl_1HP	:BOOL;//	切膜工位¶下方对中夹爪气缸1¶原点
IxS06GlampAdjustCyl_2WP	:BOOL;//	切膜工位¶下方对中夹爪气缸2¶动点
IxS06GlampAdjustCyl_2HP	:BOOL;//	切膜工位¶下方对中夹爪气缸2¶原点
IxS06GlampAdjustCyl_3WP	:BOOL;//	切膜工位¶下方对中夹爪气缸3¶动点
IxS06GlampAdjustCyl_3HP	:BOOL;//	切膜工位¶下方对中夹爪气缸3¶原点
IxS08HOZCylWP	:BOOL;//	卡片搬运工位¶水平气缸¶动点
IxS08HOZCylHP	:BOOL;//	卡片搬运工位¶水平气缸¶原点
IxShare62	:BOOL;//	备用
IxShare63	:BOOL;//	备用
IxS08VTCCyl_1WP	:BOOL;//	卡片搬运工位¶Z轴气缸1¶动点
IxS08VTCCyl_1HP	:BOOL;//	卡片搬运工位¶Z轴气缸1¶原点
IxS08VTCCyl_2WP	:BOOL;//	卡片搬运工位¶Z轴气缸2¶动点
IxS08VTCCyl_2HP	:BOOL;//	卡片搬运工位¶Z轴气缸2¶原点
IxS08Vacuum1_Output1	:BOOL;//	卡片搬运工位¶真空发生器1¶输出OUT1
IxS08Vacuum1_Output2	:BOOL;//	卡片搬运工位¶真空发生器1¶输出OUT2
IxS08Vacuum2_Output1	:BOOL;//	卡片搬运工位¶真空发生器2¶输出OUT1
IxS08Vacuum2_Output2	:BOOL;//	卡片搬运工位¶真空发生器2¶输出OUT2
IxMaintenanceSignal_1	:BOOL;//	卡片搬运工位¶离子风棒¶维护信号
IxErrorSignal_1	:BOOL;//	卡片搬运工位¶离子风棒¶异常信号
IxStartSignal	:BOOL;//	卡片搬运工位¶离子风棒¶放电信号
IxShare64	:BOOL;//	备用
IxS04Sensor1Reached	:BOOL;//	热熔工位¶深孔板¶位置1传感器
IxS04Sensor2Reached	:BOOL;//	热熔工位¶深孔板¶位置2传感器
IxS04Sensor3Reached	:BOOL;//	热熔工位¶深孔板¶位置3传感器
IxS04Sensor4Reached	:BOOL;//	热熔工位¶深孔板¶位置4传感器
IxS04AluChcekSensor1	:BOOL;//	热熔工位¶检测铝膜传感器1
IxS04AluChcekSensor2	:BOOL;//	热熔工位¶检测铝膜传感器2
IxS08CardSensor1Reached	:BOOL;//	卡片工位¶产品到位传感器1
IxS08CardSensor2Reached	:BOOL;//	卡片工位¶产品到位传感器2
IxS08CardChcekSensor1	:BOOL;//	卡片工位¶有无传感器1
IxS08CardChcekSensor2	:BOOL;//	卡片工位¶有无传感器2
IxS07CheckSensor1	:BOOL;//	NG流道¶入料口检测
IxS07CheckSensor2	:BOOL;//	NG流道¶到位传感器
IxS07CheckSensor3	:BOOL;//	NG流道¶停止传感器
IxShare65	:BOOL;//	备用
IxBufferCheckSensor1	:BOOL;//	深孔板搬运处¶缓冲位检测传感器
IxShare66	:BOOL;//	备用
IxLineEndSensor1Reached	:BOOL;//	主流线尾端¶到位检测传感器1
IxLineEndSensor2Reached	:BOOL;//	主流线尾端¶到位检测传感器2
IxLineEndCheckSensor1	:BOOL;//	主流线尾端¶有无产品传感器1
IxLineEndCheckSensor2	:BOOL;//	主流线尾端¶有无产品传感器2
IxBeltEntryCardCheckSensor1	:BOOL;//	皮带线入口处¶卡片检测传感器1
IxBeltEntryCardCheckSensor2	:BOOL;//	皮带线入口处¶卡片检测传感器2
IxBeltEntryBoxCheckSensor1	:BOOL;//	皮带线入口处¶深孔板检测传感器1
IxBeltEntryBoxCheckSensor2	:BOOL;//	皮带线入口处¶深孔板检测传感器2
IxShare71	:BOOL;//	备用
IxS06PressCyl_1WP	:BOOL;//	切膜下压气缸1动点
IxS06PressCyl_1HP	:BOOL;//	切膜下压气缸1原点
IxS06PressCyl_2WP	:BOOL;//	切膜下压气缸2动点
IxS06PressCyl_2HP	:BOOL;//	切膜下压气缸2原点
IxS06VTCCylWP	:BOOL;//	垂直切膜气缸1动点
IxS06VTCCylHP	:BOOL;//	垂直切膜气缸2原点
IxShare78	:BOOL;//	备用
IxShare79	:BOOL;//	备用
IxShare80	:BOOL;//	备用
IxShare81	:BOOL;//	备用
IxShare82	:BOOL;//	备用
IxShare83	:BOOL;//	备用
IxShare84	:BOOL;//	备用
IxShare85	:BOOL;//	备用
IxShare86	:BOOL;//	备用
IxShare87	:BOOL;//	备用
IxShare88	:BOOL;//	备用
IxShare89	:BOOL;//	备用
IxShare90	:BOOL;//	备用
IxShare91	:BOOL;//	备用
IxShare92	:BOOL;//	备用
IxShare93	:BOOL;//	备用
IxShare94	:BOOL;//	备用
QxRedLamp_1	:BOOL;//	三色灯-红灯
QxYellowLamp_1	:BOOL;//	三色灯-黄灯
QxGreenLamp_1	:BOOL;//	三色灯-绿灯
QxBuzzer_1	:BOOL;//	三色灯-蜂鸣器灯
QxHeatRelayContorl1	:BOOL;//	加热棒供电接触器1
QxHeatRelayContorl2	:BOOL;//	加热棒供电接触器2
QxMachineLamp3Contorl	:BOOL;//	日光灯控制
QxVacuum1_FeedValveControl	:BOOL;//	卡片搬运工位¶真空发生器1¶供给阀控制
QxVacuum1_BreakValveControl	:BOOL;//	卡片搬运工位¶真空发生器1¶破坏阀控制
QxVacuum2_FeedValveControl	:BOOL;//	卡片搬运工位¶真空发生器2¶供给阀控制
QxVacuum2_BreakValveControl	:BOOL;//	卡片搬运工位¶真空发生器2¶破坏阀控制
QxET02IonControlSignal1	:BOOL;//	卡片搬运工位¶离子风棒¶外部给定信号1
QxET02IonControlSignal2	:BOOL;//	卡片搬运工位¶离子风棒¶外部给定信号2
QxET02IonStopControl	:BOOL;//	卡片搬运工位¶离子风棒¶停止放电信号
QxET02IonResetControl	:BOOL;//	卡片搬运工位¶离子风棒¶复位信号
QxS09ControlValve	:BOOL;//	卡片工位离子风棒气路控制
QxS04HOZAdjustCyl_1WP	:BOOL;//	热熔工位¶上层水平调整气缸1¶动点输出
QxS04HOZAdjustCyl_1HP	:BOOL;//	热熔工位¶上层水平调整气缸1¶原点输出
QxShare75	:BOOL;//	备用
QxShare76	:BOOL;//	备用
QxS04HOZAdjustCyl_3WP	:BOOL;//	热熔工位¶下层水平调整气缸1¶动点输出
QxS04HOZAdjustCyl_3HP	:BOOL;//	热熔工位¶下层水平调整气缸1¶原点输出
QxShare77	:BOOL;//	备用
QxShare78	:BOOL;//	备用
QxS06GlampCyl_1WP	:BOOL;//	切膜工位¶前侧夹膜气缸¶动点输出
QxS06GlampCyl_1HP	:BOOL;//	切膜工位¶前侧夹膜气缸¶原点输出
QxS06GlampCyl_2WP	:BOOL;//	切膜工位¶后侧夹膜气缸¶动点输出
QxS06GlampCyl_2HP	:BOOL;//	切膜工位¶后侧夹膜气缸¶原点输出
QxS06HOZReachedCyl_1WP	:BOOL;//	切膜工位¶水平到位气缸1¶动点出输出
QxS06HOZReachedCyl_1HP	:BOOL;//	切膜工位¶水平到位气缸1¶原点出输出
QxS06HOZReachedCyl_2WP	:BOOL;//	切膜工位¶水平到位气缸2¶动点输出
QxS06HOZReachedCyl_2HP	:BOOL;//	切膜工位¶水平到位气缸2¶原点输出
QxS06HOZCyl_1WP	:BOOL;//	切膜工位¶水平切膜气缸¶动点输出
QxS06HOZCyl_1HP	:BOOL;//	切膜工位¶水平切膜气缸¶原点输出
QxS06VTCAdjustCylWP	:BOOL;//	切膜工位¶下方对中顶升气缸¶动点输出
QxS06VTCAdjustCylHP	:BOOL;//	切膜工位¶下方对中顶升气缸¶原点输出
QxS06GlampAdjustCyl_1WP	:BOOL;//	切膜工位¶下方对中夹爪气缸1¶动点输出
QxS06GlampAdjustCyl_1HP	:BOOL;//	切膜工位¶下方对中夹爪气缸1¶原点输出
QxS06GlampAdjustCyl_2WP	:BOOL;//	切膜工位¶下方对中夹爪气缸2¶动点输出
QxS06GlampAdjustCyl_2HP	:BOOL;//	切膜工位¶下方对中夹爪气缸2¶原点输出
QxS06GlampAdjustCyl_3WP	:BOOL;//	切膜工位¶下方对中夹爪气缸3¶动点输出
QxS06GlampAdjustCyl_3HP	:BOOL;//	切膜工位¶下方对中夹爪气缸3¶原点输出
QxS08HOZCylWP	:BOOL;//	卡片工位¶水平气缸¶动点输出
QxS08HOZCylHP	:BOOL;//	卡片工位¶水平气缸¶原点输出
QxS08VTCCyl_1WP	:BOOL;//	卡片工位¶Z轴气缸1¶动点输出
QxS08VTCCyl_1HP	:BOOL;//	卡片工位¶Z轴气缸1¶原点输出
QxS08VTCCyl_2WP	:BOOL;//	卡片工位¶Z轴气缸2¶动点输出
QxS08VTCCyl_2HP	:BOOL;//	卡片工位¶Z轴气缸2¶原点输出
QxS06PressCyl_1WP	:BOOL;//	切膜下压气缸1动点输出
QxS06PressCyl_1HP	:BOOL;//	切膜下压气缸1原点输出
QxS06PressCyl_2WP	:BOOL;//	切膜下压气缸2动点输出
QxS06PressCyl_2HP	:BOOL;//	切膜下压气缸2原点输出
QxS06VTCCylWP	:BOOL;//	垂直切膜气缸1动点输出
QxS06VTCCylHP	:BOOL;//	垂直切膜气缸2原点输出
QxS06BlowValve	:BOOL;//切膜工位铝膜吹气电磁阀
QxShare87	:BOOL;//	备用
QxShare88	:BOOL;//	备用
QxShare89	:BOOL;//	备用
QxShare90	:BOOL;//	备用
QxShare91	:BOOL;//	备用
QxShare92	:BOOL;//	备用
QxShare93	:BOOL;//	备用
QxShare94	:BOOL;//	备用
QxShare95	:BOOL;//	备用


IxShare100	:BOOL;//	
IxShare101	:BOOL;//	
IxShare102	:BOOL;//	
IxShare103	:BOOL;//	
IxShare104	:BOOL;//	
IxShare105	:BOOL;//	
IxShare106	:BOOL;//	
IxS01SafetyDoorReady_1	:BOOL;//	蠕动泵处安全门开关
IxShare107	:BOOL;//	
IxShare108	:BOOL;//	
IxShare109	:BOOL;//	
IxShare110	:BOOL;//	
IxShare111	:BOOL;//	
IxShare112	:BOOL;//	
IxShare113	:BOOL;//	
IxShare114	:BOOL;//	
QxLoadCell_1ZeroInput	:BOOL;//	压力传感器1清零信号
QxLoadCell_2ZeroInput	:BOOL;//	压力传感器2清零信号
QxLoadCell_3ZeroInput	:BOOL;//	压力传感器3清零信号
QxLoadCell_4ZeroInput	:BOOL;//	压力传感器4清零信号
QxLoadCell_5ZeroInput	:BOOL;//	压力传感器5清零信号
QxLoadCell_6ZeroInput	:BOOL;//	压力传感器6清零信号
QxShare165	:BOOL;//	备用
QxShare166	:BOOL;//	备用
QxShare167	:BOOL;//	备用
QxShare168	:BOOL;//	备用
QxShare169	:BOOL;//	备用
QxShare170	:BOOL;//	备用
QxShare171	:BOOL;//	备用
QxShare172	:BOOL;//	备用
QxShare173	:BOOL;//	备用
QxShare174	:BOOL;//	备用




IxLabelJobRdySignal	:BOOL;//	贴标机JOBRDY信号
IxLabelReadySignal	:BOOL;//	贴标机READY信号
IxLabelErrorSignal	:BOOL;//	贴标机ERROR信号
IxS11SensorReached1	:BOOL;//	贴标工位¶检查到位传感器1
IxS12SensorReached	:BOOL;//	标签检测工位¶检查到位传感器
IxS13SensorReached1	:BOOL;//	NG皮带线¶检测到料传感器1
IxS13SensorReached2	:BOOL;//	NG皮带线¶检测到料传感器2
IxS13SensorReached3	:BOOL;//	NG皮带线¶检测到料传感器3
IxS11HOZCylWP	:BOOL;//	贴标处推料气缸¶动点
IxS11HOZCylHP	:BOOL;//	贴标处推料气缸¶原点
IxS12HOZCyl_1WP	:BOOL;//	贴标检测工位¶推料气缸1¶动点
IxS12HOZCyl_1HP	:BOOL;//	贴标检测工位¶推料气缸1¶原点
IxS12HOZCyl_2WP	:BOOL;//	贴标检测工位¶推料气缸2¶动点
IxS12HOZCyl_2HP	:BOOL;//	贴标检测工位¶推料气缸2¶原点
IxS13HOZCyl_1WP	:BOOL;//	NG推料气缸1¶动点
IxS13HOZCyl_1HP	:BOOL;//	NG推料气缸1¶原点
IxS13HOZCyl_2WP	:BOOL;//	NG推料气缸2¶动点
IxS13HOZCyl_2HP	:BOOL;//	NG推料气缸2¶原点
IxS11SensorReached2	:BOOL;//	贴标工位¶检查到位传感器2
IxShare151	:BOOL;//	
IxShare152	:BOOL;//	
IxShare153	:BOOL;//	
IxShare154	:BOOL;//	
IxShare155	:BOOL;//	
IxShare156	:BOOL;//	
IxShare157	:BOOL;//	
IxShare158	:BOOL;//	
IxShare159	:BOOL;//	
IxShare160	:BOOL;//	
IxShare161	:BOOL;//	
IxShare162	:BOOL;//	
IxShare163	:BOOL;//	
QxMotorForward	:BOOL;//	热缩封膜出料线体¶电机正转
QxMotorStop	:BOOL;//	热缩封膜出料线体¶电机停止
QxMotorBackward	:BOOL;//	热缩封膜出料线体¶电机反转
QxMotorReserve	:BOOL;//	热缩封膜出料线体¶电机备用
QxCameraTrigger	:BOOL;//	相机触发
QxLabelStart	:BOOL;//	贴标机Start
QxLabelRibwarn	:BOOL;//	贴标机RIBWARN
QxLabelReset	:BOOL;//	贴标机RESET
QxS11HOZCylWP	:BOOL;//	贴标处推料气缸¶动点
QxS11HOZCylHP	:BOOL;//	贴标处推料气缸¶原点
QxS12HOZCyl_1WP	:BOOL;//	贴标检测工位¶推料气缸1¶动点
QxS12HOZCyl_1HP	:BOOL;//	贴标检测工位¶推料气缸1¶原点
QxS12HOZCyl_2WP	:BOOL;//	贴标检测工位¶推料气缸2¶动点
QxS12HOZCyl_2HP	:BOOL;//	贴标检测工位¶推料气缸2¶原点
QxS13HOZCyl_1WP	:BOOL;//	NG推料气缸1¶动点
QxS13HOZCyl_1HP	:BOOL;//	NG推料气缸1¶原点
QxS13HOZCyl_2WP	:BOOL;//	NG推料气缸2¶动点
QxS13HOZCyl_2HP	:BOOL;//	NG推料气缸2¶原点
QxShare150	:BOOL;//	
QxShare151	:BOOL;//	
QxShare152	:BOOL;//	
QxShare153	:BOOL;//	
QxShare154	:BOOL;//	
QxShare155	:BOOL;//	
QxShare156	:BOOL;//	
QxShare157	:BOOL;//	
QxShare158	:BOOL;//	
QxShare159	:BOOL;//	
QxShare160	:BOOL;//	
QxShare161	:BOOL;//	
QxShare162	:BOOL;//	
QxShare163	:BOOL;//	

	
	
	
	
	
	
	
	
	
	
	
	
	
	

END_VAR

// ---- POUs/40_TcpIp/40_TcpIp/TcpIpClientConstants.TcGVL
VAR_GLOBAL CONSTANT
//	PLCPRJ_RECONNECT_TIME						      : TIME := T#10MS; //连接开关延时时间;
//	PLCPRJ_SEND_CYCLE_TIME						    : TIME := T#1S;
(*	PLCPRJ_ACCEPT_POLLING_TIME					: TIME := T#1s;  not used at client side *)

//	PLCPRJ_RECEIVE_POLLING_TIME		 			  : TIME := T#1S;
//	PLCPRJ_RECEIVE_TIMEOUT						    : TIME := T#5S;
	
	(*	MAX_CLIENT_CONNECTIONS						  : UDINT(1..20) := 5; not used at client side *)
//	MAX_PLCPRJ_RXBUFFER_SIZE					    : UDINT := 300;
	
	
	
	
	MAX_CLIENT_CONNECTIONS						: DINT:=   32;(* not used at client side *)
	MAX_PLCPRJ_RXBUFFER_SIZE					: UDINT := 1000;


	PLCPRJ_RECONNECT_TIME						: TIME := T#0.5s;
	PLCPRJ_SEND_CYCLE_TIME						: TIME := T#1s;
(*	PLCPRJ_ACCEPT_POLLING_TIME					: TIME := T#1s;  not used at client side *)

	PLCPRJ_RECEIVE_POLLING_TIME		 			: TIME := T#0.5s;
	PLCPRJ_RECEIVE_TIMEOUT						: TIME := T#5s;

	(* Some project specific error codes *)
	PLCPRJ_ERROR_RECEIVE_BUFFER_OVERFLOW	: UDINT := 16#8101; (* receive buffer overflow*)
	PLCPRJ_ERROR_RECEIVE_TIMEOUT				: UDINT := 16#8102;(* receive timeout error *)

	
	
	
END_VAR

// ---- POUs/MAIN.TcPOU
PROGRAM MAIN
VAR
END_VAR

//----------------------------------------程序调用----------------------------------------------
InputLink();
S01_Loading();
S02_LidInjecting();
S03_LidChecking();
S04_AluCovering();
S05_Adjusting();
S06_Cutting();
S07_BoxCarrying();
S08_MainLine();
S09_CardCarrying();
S10_BeltCarrying();
S11_Packing();
S12_PreLine();
S13_Labeling();
S14_LabelChecking();
S15_NG();
S16_Unloading();

ControlMachine();
CallStandard();
CommWithPC();
OutputLink();
LightsTest();

END_PROGRAM

// ---- POUs/001_Station/001_Mapping/InputLink.TcPOU
PROGRAM InputLink
VAR
END_VAR

ACT_ET01();
ACT_ET02();
ACT_ET03();
ACT_ET04();

ACTION ACT_ET01:
IxSafetyRelayOK	:=	ET01_Input[1].INPUT.0	;//	安全继电器信号
IxStartButton	:=	ET01_Input[1].INPUT.1	;//	启动按钮信号
IxStopButton	:=	ET01_Input[1].INPUT.2	;//	停止按钮信号
IxResetButton	:=	ET01_Input[1].INPUT.3	;//	复位按钮信号
IxInitButton	:=	ET01_Input[1].INPUT.4	;//	初始化按钮信号
IxAutoMode	:=	ET01_Input[1].INPUT.5	;//	自动模式信号
IxManualMode	:=	ET01_Input[1].INPUT.6	;//	手动模式信号
IxAirPressure	:=	ET01_Input[1].INPUT.7	;//	上料工位¶气压检测
IxS01PositionSensor1	:=	ET01_Input[1].INPUT.8	;//	链板线深孔板¶位置1传感器
IxS01PositionSensor2	:=	ET01_Input[1].INPUT.9	;//	链板线深孔板¶位置2传感器
IxS01PositionSensor3	:=	ET01_Input[1].INPUT.10	;//	链板线深孔板¶位置3传感器
IxS01PositionSensor4	:=	ET01_Input[1].INPUT.11	;//	链板线深孔板¶位置4传感器
IxS01Sensor1Reached	:=	ET01_Input[1].INPUT.12	;//	上料工位¶到位传感器1
IxS01Sensor2Reached	:=	ET01_Input[1].INPUT.13	;//	上料工位¶到位传感器2
IxS02Sensor1Reached	:=	ET01_Input[1].INPUT.14	;//	注液工位¶到位传感器1
IxS02Sensor2Reached	:=	ET01_Input[1].INPUT.15	;//	注液工位¶到位传感器2
Ixshare2	:=	ET01_Input[2].INPUT.0	;//	备用
Ixshare3	:=	ET01_Input[2].INPUT.1	;//	备用
Ixshare4	:=	ET01_Input[2].INPUT.2	;//	备用
Ixshare5	:=	ET01_Input[2].INPUT.3	;//	备用
IxS03Sensor1Reached	:=	ET01_Input[2].INPUT.4	;//	相机工位¶到位传感器1
IxS03Sensor2Reached	:=	ET01_Input[2].INPUT.5	;//	相机工位¶到位传感器2
IxS03Sensor3Reached	:=	ET01_Input[2].INPUT.6	;//	相机工位¶到位传感器3
IxS03Sensor4Reached	:=	ET01_Input[2].INPUT.7	;//	相机工位¶到位传感器4
IxS03Sensor5Reached	:=	ET01_Input[2].INPUT.8	;//	相机工位¶到位传感器5
IxVFDErrorSignal	:=	ET01_Input[2].INPUT.9	;//	上料链板线变频器异常
Ixshare31	:=	ET01_Input[2].INPUT.10	;//	备用1
Ixshare32	:=	ET01_Input[2].INPUT.11	;//	备用2
Ixshare33	:=	ET01_Input[2].INPUT.12	;//	备用3
Ixshare34	:=	ET01_Input[2].INPUT.13	;//	备用4
IxS01SafetyDoorReady	:=	ET01_Input[2].INPUT.14	;//	上料工位安全门
IxS02SafetyDoorReady_2	:=	ET01_Input[2].INPUT.15	;//	注液工位安全门
IxS01VTCPressCyl_1WP	:=	ET01_Input[3].INPUT.0	;//	Z轴阻挡气缸1¶动点
IxS01VTCPressCyl_1HP	:=	ET01_Input[3].INPUT.1	;//	Z轴阻挡气缸1¶原点
IxS01VTCPressCyl_2WP	:=	ET01_Input[3].INPUT.2	;//	Z轴阻挡气缸2¶动点
IxS01VTCPressCyl_2HP	:=	ET01_Input[3].INPUT.3	;//	Z轴阻挡气缸2¶原点
IxS01VTCPressCyl_3WP	:=	ET01_Input[3].INPUT.4	;//	Z轴阻挡气缸3¶动点
IxS01VTCPressCyl_3HP	:=	ET01_Input[3].INPUT.5	;//	Z轴阻挡气缸3¶原点
IxS01VTCPressCyl_4WP	:=	ET01_Input[3].INPUT.6	;//	Z轴阻挡气缸4¶原点
IxS01VTCPressCyl_4HP	:=	ET01_Input[3].INPUT.7	;//	Z轴阻挡气缸4¶原点
IxS01VTCCyl_1WP	:=	ET01_Input[3].INPUT.8	;//	上料工位¶移栽Z轴气缸1¶动点
IxS01VTCCyl_1HP	:=	ET01_Input[3].INPUT.9	;//	上料工位¶移移栽Z轴气缸1¶动点
IxS01VTCCyl_2WP	:=	ET01_Input[3].INPUT.10	;//	上料工位¶移移栽Z轴气缸2¶动点
IxS01VTCCyl_2HP	:=	ET01_Input[3].INPUT.11	;//	上料工位¶移移栽Z轴气缸2¶原点
IxS02HOZAdjustCyl_1WP	:=	ET01_Input[3].INPUT.12	;//	注液工位¶上层水平调整气缸1¶动点
IxS02HOZAdjustCyl_1HP	:=	ET01_Input[3].INPUT.13	;//	注液工位¶上层水平调整气缸1¶原点
IxS02HOZAdjustCyl_2WP	:=	ET01_Input[3].INPUT.14	;//	注液工位¶上层水平调整气缸2¶动点
IxS02HOZAdjustCyl_2HP	:=	ET01_Input[3].INPUT.15	;//	注液工位¶上层水平调整气缸2¶原点
IxS02HOZAdjustCyl_3WP	:=	ET01_Input[4].INPUT.0	;//	注液工位¶下层水平调整气缸1¶动点
IxS02HOZAdjustCyl_3HP	:=	ET01_Input[4].INPUT.1	;//	注液工位¶下层水平调整气缸1¶原点点
IxS02HOZAdjustCyl_4WP	:=	ET01_Input[4].INPUT.2	;//	注液工位¶下层水平调整气缸2¶动点
IxS02HOZAdjustCyl_4HP	:=	ET01_Input[4].INPUT.3	;//	注液工位¶下层水平调整气缸2¶原点
IxS02ROTCylWP	:=	ET01_Input[4].INPUT.4	;//	注液工位¶防滴液气缸¶动点
IxS02ROTCylHP	:=	ET01_Input[4].INPUT.5	;//	注液工位¶防滴液气缸¶原点
Ixshare6	:=	ET01_Input[4].INPUT.6	;//	备用
Ixshare7	:=	ET01_Input[4].INPUT.7	;//	备用
IxS03HOZAdjustCyl_1WP	:=	ET01_Input[4].INPUT.8	;//	相机检测工位¶上层水平调整气缸1¶动点
IxS03HOZAdjustCyl_1HP	:=	ET01_Input[4].INPUT.9	;//	相机检测工位¶上层水平调整气缸1¶原点
IxS03HOZAdjustCyl_2WP	:=	ET01_Input[4].INPUT.10	;//	相机检测工位¶上层水平调整气缸2¶动点
IxS03HOZAdjustCyl_2HP	:=	ET01_Input[4].INPUT.11	;//	相机检测工位¶上层水平调整气缸2¶原点
IxS03HOZAdjustCyl_3WP	:=	ET01_Input[4].INPUT.12	;//	相机检测工位¶上层水平调整气缸3¶动点
IxS03HOZAdjustCyl_3HP	:=	ET01_Input[4].INPUT.13	;//	相机检测工位¶上层水平调整气缸3¶原点
IxS03HOZAdjustCyl_4WP	:=	ET01_Input[4].INPUT.14	;//	相机检测工位¶上层水平调整气缸4¶动点
IxS03HOZAdjustCyl_4HP	:=	ET01_Input[4].INPUT.15	;//	相机检测工位¶上层水平调整气缸4¶动点
IxS03HOZAdjustCyl_5WP	:=	ET01_Input[5].INPUT.0	;//	相机检测工位¶下层水平调整气缸1¶动点
IxS03HOZAdjustCyl_5HP	:=	ET01_Input[5].INPUT.1	;//	相机检测工位¶下层水平调整气缸1¶原点
IxS03HOZAdjustCyl_6WP	:=	ET01_Input[5].INPUT.2	;//	相机检测工位¶下层水平调整气缸2¶动点
IxS03HOZAdjustCyl_6HP	:=	ET01_Input[5].INPUT.3	;//	相机检测工位¶下层水平调整气缸2¶原点
IxS03HOZAdjustCyl_7WP	:=	ET01_Input[5].INPUT.4	;//	相机检测工位¶下层水平调整气缸3¶动点
IxS03HOZAdjustCyl_7HP	:=	ET01_Input[5].INPUT.5	;//	相机检测工位¶下层水平调整气缸3¶原点
IxS03HOZAdjustCyl_8WP	:=	ET01_Input[5].INPUT.6	;//	相机检测工位¶下层水平调整气缸4¶动点
IxS03HOZAdjustCyl_8HP	:=	ET01_Input[5].INPUT.7	;//	相机检测工位¶下层水平调整气缸4¶原点
IxErrorSignal	:=	ET01_Input[5].INPUT.8	;//	上料工位¶离子风棒¶异常信号
IxMaintenanceSignal	:=	ET01_Input[5].INPUT.9	;//	上料工位¶离子风棒¶维护信号
Ixshare9	:=	ET01_Input[5].INPUT.10	;//	备用
Ixshare10	:=	ET01_Input[5].INPUT.11	;//	备用
Ixshare11	:=	ET01_Input[5].INPUT.12	;//	备用
Ixshare12	:=	ET01_Input[5].INPUT.13	;//	备用
Ixshare13	:=	ET01_Input[5].INPUT.14	;//	备用
Ixshare14	:=	ET01_Input[5].INPUT.15	;//	备用
Ixshare15	:=	ET01_Input[6].INPUT.0	;//	备用
Ixshare16	:=	ET01_Input[6].INPUT.1	;//	备用
Ixshare17	:=	ET01_Input[6].INPUT.2	;//	备用
Ixshare18	:=	ET01_Input[6].INPUT.3	;//	备用
Ixshare19	:=	ET01_Input[6].INPUT.4	;//	备用
Ixshare20	:=	ET01_Input[6].INPUT.5	;//	备用
Ixshare21	:=	ET01_Input[6].INPUT.6	;//	备用
Ixshare22	:=	ET01_Input[6].INPUT.7	;//	备用
Ixshare23	:=	ET01_Input[6].INPUT.8	;//	备用
Ixshare24	:=	ET01_Input[6].INPUT.9	;//	备用
Ixshare25	:=	ET01_Input[6].INPUT.10	;//	备用
Ixshare26	:=	ET01_Input[6].INPUT.11	;//	备用
Ixshare27	:=	ET01_Input[6].INPUT.12	;//	备用
Ixshare28	:=	ET01_Input[6].INPUT.13	;//	备用
Ixshare29	:=	ET01_Input[6].INPUT.14	;//	备用
Ixshare30	:=	ET01_Input[6].INPUT.15	;//	备用
END_ACTION

ACTION ACT_ET02:
IxS04HOZAdjustCyl_1WP	:=	ET02_Input[1].INPUT.0	;//	热熔工位¶上层水平调整气缸1¶动点
IxS04HOZAdjustCyl_1HP	:=	ET02_Input[1].INPUT.1	;//	热熔工位¶上层水平调整气缸1¶原点
IxS04HOZAdjustCyl_2WP	:=	ET02_Input[1].INPUT.2	;//	热熔工位¶上层水平调整气缸2¶动点
IxS04HOZAdjustCyl_2HP	:=	ET02_Input[1].INPUT.3	;//	热熔工位¶上层水平调整气缸2¶原点
IxS04HOZAdjustCyl_3WP	:=	ET02_Input[1].INPUT.4	;//	热熔工位¶下层水平调整气缸1¶动点
IxS04HOZAdjustCyl_3HP	:=	ET02_Input[1].INPUT.5	;//	热熔工位¶下层水平调整气缸1¶原点
IxS04HOZAdjustCyl_4WP	:=	ET02_Input[1].INPUT.6	;//	热熔工位¶下层水平调整气缸2¶动点
IxS04HOZAdjustCyl_4HP	:=	ET02_Input[1].INPUT.7	;//	热熔工位¶下层水平调整气缸2¶原点
IxS06GlampCyl_1WP	:=	ET02_Input[1].INPUT.8	;//	切膜工位¶前侧夹膜气缸1¶动点
IxS06GlampCyl_1HP	:=	ET02_Input[1].INPUT.9	;//	切膜工位¶前侧夹膜气缸1¶原点
IxS06GlampCyl_2WP	:=	ET02_Input[1].INPUT.10	;//	切膜工位¶前侧夹膜气缸2¶动点
IxS06GlampCyl_2HP	:=	ET02_Input[1].INPUT.11	;//	切膜工位¶前侧夹膜气缸2¶原点
IxS06GlampCyl_3WP	:=	ET02_Input[1].INPUT.12	;//	切膜工位¶后侧夹膜气缸1¶动点
IxS06GlampCyl_3HP	:=	ET02_Input[1].INPUT.13	;//	切膜工位¶后侧夹膜气缸1¶原点
IxS06GlampCyl_4WP	:=	ET02_Input[1].INPUT.14	;//	切膜工位¶后侧夹膜气缸2¶动点
IxS06GlampCyl_4HP	:=	ET02_Input[1].INPUT.15	;//	切膜工位¶后侧夹膜气缸2¶原点
IxS06HOZReachedCyl_1WP	:=	ET02_Input[2].INPUT.0	;//	切膜工位¶水平到位气缸1¶动点
IxS06HOZReachedCyl_1HP	:=	ET02_Input[2].INPUT.1	;//	切膜工位¶水平到位气缸1¶原点
IxS06HOZReachedCyl_2WP	:=	ET02_Input[2].INPUT.2	;//	切膜工位¶水平到位气缸2¶动点
IxS06HOZReachedCyl_2HP	:=	ET02_Input[2].INPUT.3	;//	切膜工位¶水平到位气缸2¶原点
IxS06HOZCyl_1WP	:=	ET02_Input[2].INPUT.4	;//	切膜工位¶水平切膜气缸¶动点
IxS06HOZCyl_1HP	:=	ET02_Input[2].INPUT.5	;//	切膜工位¶水平切膜气缸¶原点
IxShare60	:=	ET02_Input[2].INPUT.6	;//	备用
IxShare61	:=	ET02_Input[2].INPUT.7	;//	备用
IxS06VTCAdjustCylWP	:=	ET02_Input[2].INPUT.8	;//	切膜工位¶下方对中顶升气缸¶动点
IxS06VTCAdjustCylHP	:=	ET02_Input[2].INPUT.9	;//	切膜工位¶下方对中顶升气缸¶原点
IxS06GlampAdjustCyl_1WP	:=	ET02_Input[2].INPUT.10	;//	切膜工位¶下方对中夹爪气缸1¶动点
IxS06GlampAdjustCyl_1HP	:=	ET02_Input[2].INPUT.11	;//	切膜工位¶下方对中夹爪气缸1¶原点
IxS06GlampAdjustCyl_2WP	:=	ET02_Input[2].INPUT.12	;//	切膜工位¶下方对中夹爪气缸2¶动点
IxS06GlampAdjustCyl_2HP	:=	ET02_Input[2].INPUT.13	;//	切膜工位¶下方对中夹爪气缸2¶原点
IxS06GlampAdjustCyl_3WP	:=	ET02_Input[2].INPUT.14	;//	切膜工位¶下方对中夹爪气缸3¶动点
IxS06GlampAdjustCyl_3HP	:=	ET02_Input[2].INPUT.15	;//	切膜工位¶下方对中夹爪气缸3¶原点
IxS08HOZCylWP	:=	ET02_Input[3].INPUT.0	;//	卡片搬运工位¶水平气缸¶动点
IxS08HOZCylHP	:=	ET02_Input[3].INPUT.1	;//	卡片搬运工位¶水平气缸¶原点
IxShare62	:=	ET02_Input[3].INPUT.2	;//	备用
IxShare63	:=	ET02_Input[3].INPUT.3	;//	备用
IxS08VTCCyl_1WP	:=	ET02_Input[3].INPUT.4	;//	卡片搬运工位¶Z轴气缸1¶动点
IxS08VTCCyl_1HP	:=	ET02_Input[3].INPUT.5	;//	卡片搬运工位¶Z轴气缸1¶原点
IxS08VTCCyl_2WP	:=	ET02_Input[3].INPUT.6	;//	卡片搬运工位¶Z轴气缸2¶动点
IxS08VTCCyl_2HP	:=	ET02_Input[3].INPUT.7	;//	卡片搬运工位¶Z轴气缸2¶原点
IxS08Vacuum1_Output1	:=	ET02_Input[3].INPUT.8	;//	卡片搬运工位¶真空发生器1¶输出OUT1
IxS08Vacuum1_Output2	:=	ET02_Input[3].INPUT.9	;//	卡片搬运工位¶真空发生器1¶输出OUT2
IxS08Vacuum2_Output1	:=	ET02_Input[3].INPUT.10	;//	卡片搬运工位¶真空发生器2¶输出OUT1
IxS08Vacuum2_Output2	:=	ET02_Input[3].INPUT.11	;//	卡片搬运工位¶真空发生器2¶输出OUT2
IxMaintenanceSignal_1	:=	ET02_Input[3].INPUT.12	;//	卡片搬运工位¶离子风棒¶维护信号
IxErrorSignal_1	:=	ET02_Input[3].INPUT.13	;//	卡片搬运工位¶离子风棒¶异常信号
IxStartSignal	:=	ET02_Input[3].INPUT.14	;//	卡片搬运工位¶离子风棒¶放电信号
IxShare64	:=	ET02_Input[3].INPUT.15	;//	备用
IxS04Sensor1Reached	:=	ET02_Input[4].INPUT.0	;//	热熔工位¶深孔板¶位置1传感器
IxS04Sensor2Reached	:=	ET02_Input[4].INPUT.1	;//	热熔工位¶深孔板¶位置2传感器
IxS04Sensor3Reached	:=	ET02_Input[4].INPUT.2	;//	热熔工位¶深孔板¶位置3传感器
IxS04Sensor4Reached	:=	ET02_Input[4].INPUT.3	;//	热熔工位¶深孔板¶位置4传感器
IxS04AluChcekSensor1	:=	ET02_Input[4].INPUT.4	;//	热熔工位¶检测铝膜传感器1
IxS04AluChcekSensor2	:=	ET02_Input[4].INPUT.5	;//	热熔工位¶检测铝膜传感器2
IxS08CardSensor1Reached	:=	ET02_Input[4].INPUT.6	;//	卡片工位¶产品到位传感器1
IxS08CardSensor2Reached	:=	ET02_Input[4].INPUT.7	;//	卡片工位¶产品到位传感器2
IxS08CardChcekSensor1	:=	ET02_Input[4].INPUT.8	;//	卡片工位¶有无传感器1
IxS08CardChcekSensor2	:=	ET02_Input[4].INPUT.9	;//	卡片工位¶有无传感器2
IxS07CheckSensor1	:=	ET02_Input[4].INPUT.10	;//	NG流道¶入料口检测
IxS07CheckSensor2	:=	ET02_Input[4].INPUT.11	;//	NG流道¶到位传感器
IxS07CheckSensor3	:=	ET02_Input[4].INPUT.12	;//	NG流道¶停止传感器
IxShare65	:=	ET02_Input[4].INPUT.13	;//	备用
IxBufferCheckSensor1	:=	ET02_Input[4].INPUT.14	;//	深孔板搬运处¶缓冲位检测传感器
IxShare66	:=	ET02_Input[4].INPUT.15	;//	备用
IxLineEndSensor1Reached	:=	ET02_Input[5].INPUT.0	;//	主流线尾端¶到位检测传感器1
IxLineEndSensor2Reached	:=	ET02_Input[5].INPUT.1	;//	主流线尾端¶到位检测传感器2
IxLineEndCheckSensor1	:=	ET02_Input[5].INPUT.2	;//	主流线尾端¶有无产品传感器1
IxLineEndCheckSensor2	:=	ET02_Input[5].INPUT.3	;//	主流线尾端¶有无产品传感器2
IxBeltEntryCardCheckSensor1	:=	ET02_Input[5].INPUT.4	;//	皮带线入口处¶卡片检测传感器1
IxBeltEntryCardCheckSensor2	:=	ET02_Input[5].INPUT.5	;//	皮带线入口处¶卡片检测传感器2
IxBeltEntryBoxCheckSensor1	:=	ET02_Input[5].INPUT.6	;//	皮带线入口处¶深孔板检测传感器1
IxBeltEntryBoxCheckSensor2	:=	ET02_Input[5].INPUT.7	;//	皮带线入口处¶深孔板检测传感器2
IxShare71	:=	ET02_Input[5].INPUT.8	;//	备用
IxS06PressCyl_1WP	:=	ET02_Input[5].INPUT.9	;//	切膜下压气缸1动点
IxS06PressCyl_1HP	:=	ET02_Input[5].INPUT.10	;//	切膜下压气缸1原点
IxS06PressCyl_2WP	:=	ET02_Input[5].INPUT.11	;//	切膜下压气缸2动点
IxS06PressCyl_2HP	:=	ET02_Input[5].INPUT.12	;//	切膜下压气缸2原点
IxS06VTCCylWP	:=	ET02_Input[5].INPUT.13	;//	垂直切膜气缸1动点
IxS06VTCCylHP	:=	ET02_Input[5].INPUT.14	;//	垂直切膜气缸2原点
IxShare78	:=	ET02_Input[5].INPUT.15	;//	备用
IxShare79	:=	ET02_Input[6].INPUT.0	;//	备用
IxShare80	:=	ET02_Input[6].INPUT.1	;//	备用
IxShare81	:=	ET02_Input[6].INPUT.2	;//	备用
IxShare82	:=	ET02_Input[6].INPUT.3	;//	备用
IxShare83	:=	ET02_Input[6].INPUT.4	;//	备用
IxShare84	:=	ET02_Input[6].INPUT.5	;//	备用
IxShare85	:=	ET02_Input[6].INPUT.6	;//	备用
IxShare86	:=	ET02_Input[6].INPUT.7	;//	备用
IxShare87	:=	ET02_Input[6].INPUT.8	;//	备用
IxShare88	:=	ET02_Input[6].INPUT.9	;//	备用
IxShare89	:=	ET02_Input[6].INPUT.10	;//	备用
IxShare90	:=	ET02_Input[6].INPUT.11	;//	备用
IxShare91	:=	ET02_Input[6].INPUT.12	;//	备用
IxShare92	:=	ET02_Input[6].INPUT.13	;//	备用
IxShare93	:=	ET02_Input[6].INPUT.14	;//	备用
IxShare94	:=	ET02_Input[6].INPUT.15	;//	备用
END_ACTION

ACTION ACT_ET03:
IxShare100	:=	ET03_Input[1].INPUT.0	;//	备用
IxShare101	:=	ET03_Input[1].INPUT.1	;//	备用
IxShare102	:=	ET03_Input[1].INPUT.2	;//	备用
IxShare103	:=	ET03_Input[1].INPUT.3	;//	备用
IxShare104	:=	ET03_Input[1].INPUT.4	;//	备用
IxShare105	:=	ET03_Input[1].INPUT.5	;//	备用
IxShare106	:=	ET03_Input[1].INPUT.6	;//	备用
IxS01SafetyDoorReady_1	:=	ET03_Input[1].INPUT.7;//	蠕动泵处安全门开关
IxShare107	:=	ET03_Input[1].INPUT.8	;//	备用
IxShare108	:=	ET03_Input[1].INPUT.9	;//	备用
IxShare109	:=	ET03_Input[1].INPUT.10	;//	备用
IxShare110	:=	ET03_Input[1].INPUT.11	;//	备用
IxShare111	:=	ET03_Input[1].INPUT.12	;//	备用
IxShare112	:=	ET03_Input[1].INPUT.13	;//	备用
IxShare113	:=	ET03_Input[1].INPUT.14	;//	备用
IxShare114	:=	ET03_Input[1].INPUT.15	;//	备用
END_ACTION

ACTION ACT_ET04:
IxLabelJobRdySignal	:=	ET04_Input[1].INPUT.0	;//	贴标机JOBRDY信号
IxLabelReadySignal	:=	ET04_Input[1].INPUT.1	;//	贴标机READY信号
IxLabelErrorSignal	:=	ET04_Input[1].INPUT.2	;//	贴标机ERROR信号
IxS11SensorReached1	:=	ET04_Input[1].INPUT.3	;//	贴标工位¶检查到位传感器
IxS12SensorReached	:=	ET04_Input[1].INPUT.4	;//	标签检测工位¶检查到位传感器
IxS13SensorReached1	:=	ET04_Input[1].INPUT.5	;//	NG皮带线¶检测到料传感器1
IxS13SensorReached2	:=	ET04_Input[1].INPUT.6	;//	NG皮带线¶检测到料传感器2
IxS13SensorReached3	:=	ET04_Input[1].INPUT.7	;//	NG皮带线¶检测到料传感器3
IxS11HOZCylWP	:=	ET04_Input[1].INPUT.8	;//	贴标处推料气缸¶动点
IxS11HOZCylHP	:=	ET04_Input[1].INPUT.9	;//	贴标处推料气缸¶原点
IxS12HOZCyl_1WP	:=	ET04_Input[1].INPUT.10	;//	贴标检测工位¶推料气缸1¶动点
IxS12HOZCyl_1HP	:=	ET04_Input[1].INPUT.11	;//	贴标检测工位¶推料气缸1¶原点
IxS12HOZCyl_2WP	:=	ET04_Input[1].INPUT.12	;//	贴标检测工位¶推料气缸2¶动点
IxS12HOZCyl_2HP	:=	ET04_Input[1].INPUT.13	;//	贴标检测工位¶推料气缸2¶原点
IxS13HOZCyl_1WP	:=	ET04_Input[1].INPUT.14	;//	NG推料气缸1¶动点
IxS13HOZCyl_1HP	:=	ET04_Input[1].INPUT.15	;//	NG推料气缸1¶原点
IxS13HOZCyl_2WP	:=	ET04_Input[2].INPUT.0	;//	NG推料气缸2¶动点
IxS13HOZCyl_2HP	:=	ET04_Input[2].INPUT.1	;//	NG推料气缸2¶原点
IxS11SensorReached2	:=	ET04_Input[2].INPUT.2	;//	贴标工位¶检查到位传感器2
IxShare151	:=	ET04_Input[2].INPUT.3	;//	备用
IxShare152	:=	ET04_Input[2].INPUT.4	;//	备用
IxShare153	:=	ET04_Input[2].INPUT.5	;//	备用
IxShare154	:=	ET04_Input[2].INPUT.6	;//	备用
IxShare155	:=	ET04_Input[2].INPUT.7	;//	备用
IxShare156	:=	ET04_Input[2].INPUT.8	;//	备用
IxShare157	:=	ET04_Input[2].INPUT.9	;//	备用
IxShare158	:=	ET04_Input[2].INPUT.10	;//	备用
IxShare159	:=	ET04_Input[2].INPUT.11	;//	备用
IxShare160	:=	ET04_Input[2].INPUT.12	;//	备用
IxShare161	:=	ET04_Input[2].INPUT.13	;//	备用
IxShare162	:=	ET04_Input[2].INPUT.14	;//	备用
IxShare163	:=	ET04_Input[2].INPUT.15	;//	备用
END_ACTION

END_PROGRAM

// ---- POUs/001_Station/S01_Loading.TcPOU
PROGRAM S01_Loading
VAR
	//工站
	station					: REFERENCE TO FB_Station:=fbstation[1];
	//气缸
		fbVTCPressCyl_1	:REFERENCE TO FB_Cylinder:=fbCylinder[1];	//	链板线-下压气缸1
		fbVTCPressCyl_2	:REFERENCE TO FB_Cylinder:=fbCylinder[2];	//	链板线-下压气缸2
		fbVTCPressCyl_3	:REFERENCE TO FB_Cylinder:=fbCylinder[3];	//	链板线-下压气缸3
		fbVTCPressCyl_4	:REFERENCE TO FB_Cylinder:=fbCylinder[4];	//	链板线-下压气缸4
		fbVTCCyl_1	:REFERENCE TO FB_Cylinder:=fbCylinder[5];	//	移栽机构-Z轴气缸1
		fbVTCCyl_2	:REFERENCE TO FB_Cylinder:=fbCylinder[6];	//	移栽机构-Z轴气缸2
//链板线
		fbFlowLine:FB_FlowLine;	
		
	//伺服
		fbXAxisMove	 :REFERENCE TO FB_Axis:=fbAxis[1];	//	移栽上料X轴伺服
		fbYAxisMove	 :REFERENCE TO FB_Axis:=fbAxis[2];	//	移栽上料Y轴伺服
	//电动夹爪
		fbClamp_1:	 REFERENCE TO FB_ERG_20_Modbus:=fbERG_20_Modbus[1];
		fbClamp_2:	 REFERENCE TO FB_ERG_20_Modbus:=fbERG_20_Modbus[2];
		
		ERG_20C_1	:		 REFERENCE TO FB_ERG_20C:=fbERG[1];
		ERG_20C_2	:		 REFERENCE TO FB_ERG_20C:=fbERG[2];
		
	//相机
		 Camera   : 	 REFERENCE TO FB_Camera:=fbCamera[1]; 
	//延时
	arTonDelay :ARRAY[1..20] OF TON;
	//返回值
	UdiReturnValue :ARRAY[1..20] OF UDINT;
	//本地过程数据
	arProcessDataStation : ARRAY [1..2] OF DUT_MainlineFixture;
	//过程标志位
	xFlowLineReady:BOOL;//连班线准备流程完成信号
	xTakeBoxPremit:BOOL;//允许链板线执行下一循环
	//过程记录
	tsModuleProcess:ARRAY[1..gc_ModuleProNo] OF DUT_Process;
	xClearModuleProcessDone:BOOL;
	bClearProcessStep	:BYTE;
	
	
	i: INT;
	xFlowLineStart: BOOL;//链板线启动信号
	bFlowLineStep: BYTE;
	xFlowLineReadyCmd: BOOL;//连班线准备指令
	arFlowLineReachedSensor: ARRAY[1..4] OF BOOL;//链板线到位传感器
	_FirstFlag: ARRAY[1..10] OF BOOL;
	MachineInitR_TRIG:R_TRIG;

	// 程序循环
	bCounter: BYTE;
	// 上料工位到位传感器
	xLoadingReachedSensor: ARRAY[1..2] of bool;
	// 报警标志位
	_AlarmDisable: BOOL;
	// X轴放料循环
	bXCounter: BYTE;
	//夹爪有产品信号
	arClampHavePart :ARRAY[1..2] OF BOOL;
	iClearProcessStep: INT;
	// //首次循环
	_FirstCycle: ARRAY[1..10] of bool;
	//下压气缸原点传感器
	arVTCPressCylHPSensor:ARRAY[1..4] OF BOOL;
	//Y轴去放料位还是放料补偿位
	ariPosNum:ARRAY[1..2] OF INT;
	//下压气缸动点传感器
	arVTCPressCylWPSensor:ARRAY[1..4] OF BOOL;
	test: ARRAY[1..4]OF BOOL;
	// 步骤
	itestStep: INT;
	// 按钮
	xtestbutton: BOOL;
END_VAR

A_Input();
Alarm();
Delay();
FlowAuto();
FlowInit();
//FlowAuto_1();
//FlowInit_1();
FlowLine();
General();
ILC();
TipAuto();
TipManual();
Z_Output();

ACTION A_Input:
//气缸
fbVTCPressCyl_1.xWP_Sensor	:=
arVTCPressCylWPSensor[1]		:=	IxS01VTCPressCyl_1WP 	;
fbVTCPressCyl_1.xHP_Sensor	:=
arVTCPressCylHPSensor[1]		:=	IxS01VTCPressCyl_1HP	;
fbVTCPressCyl_2.xWP_Sensor	:=	
arVTCPressCylWPSensor[2]		:=	IxS01VTCPressCyl_2WP	;
fbVTCPressCyl_2.xHP_Sensor	:=
arVTCPressCylHPSensor[2]		:=	IxS01VTCPressCyl_2HP	;
fbVTCPressCyl_3.xWP_Sensor	:=	
arVTCPressCylWPSensor[3]		:=IxS01VTCPressCyl_3WP	;
fbVTCPressCyl_3.xHP_Sensor	:=
arVTCPressCylHPSensor[3]		:=	IxS01VTCPressCyl_3HP	;
fbVTCPressCyl_4.xWP_Sensor	:=	
arVTCPressCylWPSensor[4]		:=IxS01VTCPressCyl_4WP	;
fbVTCPressCyl_4.xHP_Sensor	:=
arVTCPressCylHPSensor[4]		:=IxS01VTCPressCyl_4HP	;
fbVTCCyl_1.xWP_Sensor	:=	IxS01VTCCyl_1WP	;
fbVTCCyl_1.xHP_Sensor	:=	IxS01VTCCyl_1HP	;
fbVTCCyl_2.xWP_Sensor	:=	IxS01VTCCyl_2WP	;
fbVTCCyl_2.xHP_Sensor	:=	IxS01VTCCyl_2HP	;

//链板线传感器
arFlowLineReachedSensor[1]:=IxS01PositionSensor2;
arFlowLineReachedSensor[2]:=IxS01PositionSensor1;
arFlowLineReachedSensor[3]:=IxS01PositionSensor4;
arFlowLineReachedSensor[4]:=IxS01PositionSensor3;
//上料工位传感器
xLoadingReachedSensor[1]:=IxS01Sensor2Reached;
xLoadingReachedSensor[2]:=IxS01Sensor1Reached;
END_ACTION

ACTION Alarm:
//
station.adwAlarm[1].00:=station.xInitTimeout;	  //S01 初始化超时
//station.adwAlarm[1].01:= //S01链板线上料位置1相机检测到深孔板放反，请检查
//station.adwAlarm[1].02:=//S01链板线上料位置2相机检测到深放反，请检查
//station.adwAlarm[1].03:=//S01链板线上料位置3相机检测到深孔板放反，请检查
//station.adwAlarm[1].04:=//S01链板线上料位置4相机检测到深孔板放反，请检查
station.adwAlarm[1].05	:=	fbClamp_1.eErrorID>24	;//	S01电动夹爪1报错，请检查
station.adwAlarm[1].06	:=	fbClamp_2.eErrorID>24	;//	S01电动夹爪2报错，请检查
//station.adwAlarm[1].07	:=	fbVTCPressCyl_1.xHP_Off 	;//	S01链板线-下压气缸1原点未到位
//station.adwAlarm[1].08	:=	fbVTCPressCyl_1.xWP_Off 	;//	S01链板线-下压气缸1动点未到位
//station.adwAlarm[1].09	:=	fbVTCPressCyl_2.xHP_Off	;//	S01链板线-下压气缸2原点未到位
//station.adwAlarm[1].10	:=	fbVTCPressCyl_2.xWP_Off	;//	S01链板线-下压气缸2动点未到位
//station.adwAlarm[1].11	:=	fbVTCPressCyl_3.xHP_Off	;//	S01链板线-下压气缸3原点未到位
//station.adwAlarm[1].12	:=	fbVTCPressCyl_3.xWP_Off	;//	S01链板线-下压气缸3动点未到位
//station.adwAlarm[1].13	:=	fbVTCPressCyl_4.xHP_Off	;//	S01链板线-下压气缸4原点未到位
//station.adwAlarm[1].14	:=	fbVTCPressCyl_4.xWP_Off	;//	S01链板线-下压气缸4动点未到位
station.adwAlarm[1].15	:=	fbVTCCyl_1.xHP_Off 	;//	S01移栽机构-Z轴气缸1原点未到位
station.adwAlarm[1].16	:=	fbVTCCyl_1.xWP_Off	;//	S01移栽机构-Z轴气缸1动点未到位
station.adwAlarm[1].17	:=	fbVTCCyl_2.xHP_Off 	;//	S01移栽机构-Z轴气缸2原点未到位
station.adwAlarm[1].18	:=	fbVTCCyl_2.xWP_Off	;//	S01移栽机构-Z轴气缸2动点未到位
station.adwAlarm[1].19	:=	fbXAxisMove.xError	;//	S01移栽上料X轴伺服报错
station.adwAlarm[1].20	:=	fbXAxisMove.xNotPowerOn	;//	S01移栽上料X轴伺服未使能
station.adwAlarm[1].21	:=	fbXAxisMove.xMoveTimeout	;//	S01移栽上料X轴伺服移动超时
station.adwAlarm[1].22	:=	fbYAxisMove.xError	;//	S01移栽上料Y轴伺服报错
station.adwAlarm[1].23	:=	fbYAxisMove.xNotPowerOn	;//	S01移栽上料Y轴伺服未使能
station.adwAlarm[1].24	:=	fbYAxisMove.xMoveTimeout	;//	S01移栽上料Y轴伺服移动超时
//station.adwAlarm[1].25	:=	fbFlowLine.xQError	;			//	S01移栽上料链板线报错

//station.adwAlarm[1].26:= //S01链板线上料位置1相机检测到深孔板放反，请检查
//station.adwAlarm[1].27:=//S01链板线上料位置2相机检测到深放反，请检查
//station.adwAlarm[1].28:=//S01链板线上料位置3相机检测到深孔板放反，请检查
//station.adwAlarm[1].29:=//S01链板线上料位置4相机检测到深孔板放反，请检查
//station.adwAlarm[1].30	:=	TRUE;//	S01上料工位-相机拍照超时，请检查
//station.adwAlarm[1].31	:=	TRUE;//	S01上料工位-链板线运行超时,请复位
END_ACTION

ACTION Delay:
arTonDelay[01](IN:= , PT:=T#0.1S , Q=> , ET=> );
//arTonDelay[02](IN:=  , PT:=T#1S , Q=> , ET=> );*)//链板线程序使用
//arTonDelay[03](IN:=   , PT:=T#1S , Q=> , ET=> );//已使用
arTonDelay[04](IN:= , PT:=T#0.1S , Q=> , ET=> );
arTonDelay[05](IN:= , PT:=T#0.1S , Q=> , ET=> );
arTonDelay[06](IN:= , PT:=T#0.1S , Q=> , ET=> );
arTonDelay[07](IN:= , PT:=T#0.1S , Q=> , ET=> );
arTonDelay[08](IN:= NOT fbXAxisMove.xbusy , PT:=T#0.1S , Q=> , ET=> );//TipAuto使用
arTonDelay[09](IN:= NOT fbYAxisMove.xbusy, PT:=T#0.1S , Q=> , ET=> );//TipAuto使用
END_ACTION

ACTION FlowAuto:

//-----------------------------------------初始化是否完成判断----------------------------------------------
IF NOT station.xInitDone THEN
 	station.iStepAuto:=0;
 	station.xDone:=FALSE;
ELSIF station.xRunning  OR 
//(tsModuleProcess[1].xProcessStarted AND  NOT tsModuleProcess[1].xProcessCompleted)  OR//相机拍照流程
(	tsModuleProcess[bCounter+1].xProcessStarted AND  NOT tsModuleProcess[bCounter+1].xProcessCompleted)  OR //电动夹爪夹取流程
(tsModuleProcess[bCounter+3].xProcessStarted AND  NOT tsModuleProcess[bCounter+3].xProcessCompleted)  OR //孔板翻转流程流程
(	tsModuleProcess[bXCounter+5].xProcessStarted AND NOT 	tsModuleProcess[bXCounter+5].xProcessCompleted) //电动夹爪松开流程
THEN
//-----------------------------------------动作步骤--------------------------------------------------------
CASE station.iStepAuto OF	  
	0: //----Home Step，等待启动----
		IF station.xDisabled 
			AND station.xCanRun 
			AND NOT fbMachine[1].xStopped 
			AND NOT station.xSingleRunning 
		THEN
			station.xDone:=TRUE;
		END_IF
		IF  station.xSingleRunning 
			OR station.xCanRun 
			//AND NOT station.xDone 
			AND NOT station.xDisabled 
			AND NOT fbMachine[1].xStopped
		THEN
			station.xCycleEnable:=TRUE;
			//station.xDone:= FALSE;  
			station.iStepAuto:= 10;
		END_IF
	10://复位
			Camera.xlInit:=TRUE;
			FOR  i:=1 TO  4 BY  1 DO
		 		sCamera_To_Plc.iS01Result[i]:=0;
			END_FOR
			MEMSET(ADR(arProcessDataStation[1]),0,SIZEOF(arProcessDataStation[1]));
			MEMSET(ADR(arProcessDataStation[2]),0,SIZEOF(arProcessDataStation[2]));
		
